LIN {X 0,Y 230.328,Z 772.05,A -85,B 0,C 180,E1 -20406.395,E2 -20406.395} C_VEL
LIN {X 0,Y 229.138,Z 759.993,A -85,B 0,C 180,E1 -20407.932,E2 -20407.932} C_VEL
LIN {X 0,Y 227.349,Z 746.527,A -85,B 0,C 180,E1 -20409.296,E2 -20409.296} C_VEL
LIN {X 0,Y 224.848,Z 732.445,A -85,B 0,C 180,E1 -20410.367,E2 -20410.367} C_VEL
LIN {X 0,Y 224.753,Z 731.518,A -85,B 0,C 180,E1 -20410.477,E2 -20410.477} C_VEL
LIN {X 0,Y 225.974,Z 721.97,A -85,B 0,C 180,E1 -20414.606,E2 -20414.606} C_VEL
LIN {X 0,Y 227.437,Z 711.151,A -85,B 0,C 180,E1 -20419.316,E2 -20419.316} C_VEL
LIN {X 0,Y 227.799,Z 707.066,A -85,B 0,C 180,E1 -20421.127,E2 -20421.127} C_VEL
LIN {X 0,Y 227.341,Z 701.42,A -85,B 0,C 180,E1 -20423.79,E2 -20423.79} C_VEL
LIN {X 0,Y 225.605,Z 691.076,A -85,B 0,C 180,E1 -20428.938,E2 -20428.938} C_VEL
LIN {X 0,Y 224.604,Z 685.498,A -85,B 0,C 180,E1 -20431.794,E2 -20431.794} C_VEL
LIN {X 0,Y 221.937,Z 675.451,A -85,B 0,C 180,E1 -20437.278,E2 -20437.278} C_VEL
LIN {X 0,Y 221.276,Z 672.918,A -85,B 0,C 180,E1 -20438.793,E2 -20438.793} C_VEL
LIN {X 0,Y 221.288,Z 673.134,A -85,B 0,C 180,E1 -20439.08,E2 -20439.08} C_VEL
LIN {X 0,Y 225.275,Z 684.524,A -85,B 0,C 180,E1 -20440.789,E2 -20440.789} C_VEL
LIN {X 0,Y 228.656,Z 695.212,A -85,B 0,C 180,E1 -20442.651,E2 -20442.651} C_VEL
LIN {X 0,Y 231.416,Z 705.742,A -85,B 0,C 180,E1 -20444.736,E2 -20444.736} C_VEL
LIN {X 0,Y 231.578,Z 706.808,A -85,B 0,C 180,E1 -20444.95,E2 -20444.95} C_VEL
LIN {X 0,Y 229.57,Z 717.919,A -85,B 0,C 180,E1 -20447.138,E2 -20447.138} C_VEL
LIN {X 0,Y 227.893,Z 726.962,A -85,B 0,C 180,E1 -20449.361,E2 -20449.361} C_VEL
LIN {X 0,Y 226.116,Z 735.343,A -85,B 0,C 180,E1 -20451.9,E2 -20451.9} C_VEL
LIN {X 0,Y 224.502,Z 742.894,A -85,B 0,C 180,E1 -20454.792,E2 -20454.792} C_VEL
LIN {X 0,Y 223.525,Z 747.733,A -85,B 0,C 180,E1 -20457.098,E2 -20457.098} C_VEL
LIN {X 0,Y 222.474,Z 753.098,A -85,B 0,C 180,E1 -20460.362,E2 -20460.362} C_VEL
LIN {X 0,Y 221.947,Z 755.831,A -85,B 0,C 180,E1 -20462.569,E2 -20462.569} C_VEL
LIN {X 0,Y 221.622,Z 757.987,A -85,B 0,C 180,E1 -20464.808,E2 -20464.808} C_VEL
LIN {X 0,Y 221.54,Z 759.729,A -85,B 0,C 180,E1 -20467.526,E2 -20467.526} C_VEL
LIN {X 0,Y 221.871,Z 760.631,A -85,B 0,C 180,E1 -20470.516,E2 -20470.516} C_VEL
LIN {X 0,Y 222.756,Z 760.329,A -85,B 0,C 180,E1 -20473.957,E2 -20473.957} C_VEL
LIN {X 0,Y 223.638,Z 759.356,A -85,B 0,C 180,E1 -20476.286,E2 -20476.286} C_VEL
LIN {X 0,Y 225.52,Z 756.419,A -85,B 0,C 180,E1 -20479.898,E2 -20479.898} C_VEL
LIN {X 0,Y 227.153,Z 753.336,A -85,B 0,C 180,E1 -20482.401,E2 -20482.401} C_VEL
LIN {X 0,Y 229.082,Z 749.336,A -85,B 0,C 180,E1 -20484.857,E2 -20484.857} C_VEL
LIN {X 0,Y 231.336,Z 744.272,A -85,B 0,C 180,E1 -20487.28,E2 -20487.28} C_VEL
LIN {X 0,Y 233.865,Z 738.05,A -85,B 0,C 180,E1 -20489.641,E2 -20489.641} C_VEL
LIN {X 0,Y 236.623,Z 730.403,A -85,B 0,C 180,E1 -20491.971,E2 -20491.971} C_VEL
LIN {X 0,Y 239.577,Z 721.408,A -85,B 0,C 180,E1 -20494.152,E2 -20494.152} C_VEL
LIN {X 0,Y 239.995,Z 719.96,A -85,B 0,C 180,E1 -20494.456,E2 -20494.456} C_VEL
LIN {X 0,Y 239.14,Z 713.976,A -85,B 0,C 180,E1 -20496.166,E2 -20496.166} C_VEL
LIN {X 0,Y 236.776,Z 705.016,A -85,B 0,C 180,E1 -20498.678,E2 -20498.678} C_VEL
LIN {X 0,Y 233.522,Z 696.191,A -85,B 0,C 180,E1 -20501.124,E2 -20501.124} C_VEL
LIN {X 0,Y 229.459,Z 687.704,A -85,B 0,C 180,E1 -20503.542,E2 -20503.542} C_VEL
LIN {X 0,Y 226.423,Z 682.123,A -85,B 0,C 180,E1 -20505.163,E2 -20505.163} C_VEL
LIN {X 0,Y 224.367,Z 678.912,A -85,B 0,C 180,E1 -20506.178,E2 -20506.178} C_VEL
LIN {X 0,Y 223.667,Z 677.621,A -85,B 0,C 180,E1 -20506.542,E2 -20506.542} C_VEL
LIN {X 0,Y 221.78,Z 675.276,A -85,B 0,C 180,E1 -20507.417,E2 -20507.417} C_VEL
LIN {X 0,Y 221.062,Z 672.945,A -85,B 0,C 180,E1 -20507.958,E2 -20507.958} C_VEL
LIN {X 0,Y 221.24,Z 672.924,A -85,B 0,C 180,E1 -20510.861,E2 -20510.861} C_VEL
LIN {X 0,Y 221.293,Z 672.907,A -85,B 0,C 180,E1 -20512.702,E2 -20512.702} C_VEL
LIN {X 0,Y 221.516,Z 672.886,A -85,B 0,C 180,E1 -20518.182,E2 -20518.182} C_VEL
LIN {X 0,Y 221.516,Z 672.88,A -85,B 0,C 180,E1 -20521.818,E2 -20521.818} C_VEL
LIN {X 0,Y 221.309,Z 672.918,A -85,B 0,C 180,E1 -20527.298,E2 -20527.298} C_VEL
LIN {X 0,Y 221.11,Z 672.944,A -85,B 0,C 180,E1 -20530.995,E2 -20530.995} C_VEL
LIN {X 0,Y 221.02,Z 672.944,A -85,B 0,C 180,E1 -20536.63,E2 -20536.63} C_VEL
LIN {X 0,Y 220.948,Z 673.087,A -85,B 0,C 180,E1 -20541.947,E2 -20541.947} C_VEL
LIN {X 0,Y 221.61,Z 676.139,A -85,B 0,C 180,E1 -20546.359,E2 -20546.359} C_VEL
LIN {X 0,Y 222.496,Z 680.424,A -85,B 0,C 180,E1 -20551.476,E2 -20551.476} C_VEL
LIN {X 0,Y 223.333,Z 683.935,A -85,B 0,C 180,E1 -20555.095,E2 -20555.095} C_VEL
LIN {X 0,Y 224.157,Z 688.047,A -85,B 0,C 180,E1 -20558.834,E2 -20558.834} C_VEL
LIN {X 0,Y 224.93,Z 692.081,A -85,B 0,C 180,E1 -20562.168,E2 -20562.168} C_VEL
LIN {X 0,Y 224.511,Z 693.459,A -85,B 0,C 180,E1 -20563.107,E2 -20563.107} C_VEL
LIN {X 0,Y 222.094,Z 696.117,A -85,B 0,C 180,E1 -20564.563,E2 -20564.563} C_VEL
LIN {X 0,Y 219.629,Z 698.835,A -85,B 0,C 180,E1 -20566.046,E2 -20566.046} C_VEL
LIN {X 0,Y 219.18,Z 700.319,A -85,B 0,C 180,E1 -20567.012,E2 -20567.012} C_VEL
LIN {X 0,Y 219.597,Z 703.203,A -85,B 0,C 180,E1 -20569.033,E2 -20569.033} C_VEL
LIN {X 0,Y 220.976,Z 707.443,A -85,B 0,C 180,E1 -20569.757,E2 -20569.757} C_VEL
LIN {X 0,Y 221.732,Z 709.798,A -85,B 0,C 180,E1 -20570.174,E2 -20570.174} C_VEL
LIN {X 0,Y 224.611,Z 722.385,A -85,B 0,C 180,E1 -20572.15,E2 -20572.15} C_VEL
LIN {X 0,Y 226.492,Z 736.93,A -85,B 0,C 180,E1 -20574.426,E2 -20574.426} C_VEL
LIN {X 0,Y 226.964,Z 748.451,A -85,B 0,C 180,E1 -20576.31,E2 -20576.31} C_VEL
LIN {X 0,Y 226.482,Z 760.232,A -85,B 0,C 180,E1 -20578.422,E2 -20578.422} C_VEL
LIN {X 0,Y 225.182,Z 771.012,A -85,B 0,C 180,E1 -20580.589,E2 -20580.589} C_VEL
LIN {X 0,Y 223.216,Z 780.783,A -85,B 0,C 180,E1 -20582.835,E2 -20582.835} C_VEL
LIN {X 0,Y 221.932,Z 786.81,A -85,B 0,C 180,E1 -20584.438,E2 -20584.438} C_VEL
LIN {X 0,Y 221.121,Z 796.098,A -85,B 0,C 180,E1 -20585.844,E2 -20585.844} C_VEL
LIN {X 0,Y 218.923,Z 807.176,A -85,B 0,C 180,E1 -20587.838,E2 -20587.838} C_VEL
LIN {X 0,Y 217.03,Z 816.687,A -85,B 0,C 180,E1 -20590.013,E2 -20590.013} C_VEL
LIN {X 0,Y 215.729,Z 823.747,A -85,B 0,C 180,E1 -20591.971,E2 -20591.971} C_VEL
LIN {X 0,Y 214.068,Z 831.966,A -85,B 0,C 180,E1 -20594.772,E2 -20594.772} C_VEL
LIN {X 0,Y 212.846,Z 838.572,A -85,B 0,C 180,E1 -20597.606,E2 -20597.606} C_VEL
LIN {X 0,Y 212.118,Z 843.817,A -85,B 0,C 180,E1 -20600.463,E2 -20600.463} C_VEL
LIN {X 0,Y 211.718,Z 847.843,A -85,B 0,C 180,E1 -20603.327,E2 -20603.327} C_VEL
LIN {X 0,Y 211.566,Z 850.772,A -85,B 0,C 180,E1 -20606.19,E2 -20606.19} C_VEL
LIN {X 0,Y 211.618,Z 852.149,A -85,B 0,C 180,E1 -20608.096,E2 -20608.096} C_VEL
LIN {X 0,Y 211.718,Z 853.102,A -85,B 0,C 180,E1 -20609.999,E2 -20609.999} C_VEL
LIN {X 0,Y 211.582,Z 853.643,A -85,B 0,C 180,E1 -20611.902,E2 -20611.902} C_VEL
LIN {X 0,Y 211.507,Z 853.693,A -85,B 0,C 180,E1 -20614.548,E2 -20614.548} C_VEL
LIN {X 0,Y 211.769,Z 852.796,A -85,B 0,C 180,E1 -20617.627,E2 -20617.627} C_VEL
LIN {X 0,Y 212.753,Z 850.263,A -85,B 0,C 180,E1 -20621.431,E2 -20621.431} C_VEL
LIN {X 0,Y 213.945,Z 847.262,A -85,B 0,C 180,E1 -20624.262,E2 -20624.262} C_VEL
LIN {X 0,Y 215.748,Z 843.249,A -85,B 0,C 180,E1 -20627.047,E2 -20627.047} C_VEL
LIN {X 0,Y 218.124,Z 838.128,A -85,B 0,C 180,E1 -20629.773,E2 -20629.773} C_VEL
LIN {X 0,Y 221.012,Z 831.011,A -85,B 0,C 180,E1 -20632.753,E2 -20632.753} C_VEL
LIN {X 0,Y 224.587,Z 822.54,A -85,B 0,C 180,E1 -20635.484,E2 -20635.484} C_VEL
LIN {X 0,Y 227.743,Z 814.382,A -85,B 0,C 180,E1 -20637.572,E2 -20637.572} C_VEL
LIN {X 0,Y 231.693,Z 803.348,A -85,B 0,C 180,E1 -20639.781,E2 -20639.781} C_VEL
LIN {X 0,Y 234.219,Z 792.567,A -85,B 0,C 180,E1 -20641.674,E2 -20641.674} C_VEL
LIN {X 0,Y 236.122,Z 782.049,A -85,B 0,C 180,E1 -20643.197,E2 -20643.197} C_VEL
LIN {X 0,Y 236.663,Z 772.17,A -85,B 0,C 180,E1 -20644.583,E2 -20644.583} C_VEL
LIN {X 0,Y 235.936,Z 759.615,A -85,B 0,C 180,E1 -20646.321,E2 -20646.321} C_VEL
LIN {X 0,Y 233.902,Z 747.598,A -85,B 0,C 180,E1 -20648.007,E2 -20648.007} C_VEL
LIN {X 0,Y 231.196,Z 736.83,A -85,B 0,C 180,E1 -20649.669,E2 -20649.669} C_VEL
LIN {X 0,Y 232.487,Z 726.541,A -85,B 0,C 180,E1 -20652.996,E2 -20652.996} C_VEL
LIN {X 0,Y 231.85,Z 720.918,A -85,B 0,C 180,E1 -20655.797,E2 -20655.797} C_VEL
LIN {X 0,Y 231.289,Z 715.047,A -85,B 0,C 180,E1 -20659.432,E2 -20659.432} C_VEL
LIN {X 0,Y 231.206,Z 712.321,A -85,B 0,C 180,E1 -20661.455,E2 -20661.455} C_VEL
LIN {X 0,Y 230.48,Z 709.689,A -85,B 0,C 180,E1 -20664.594,E2 -20664.594} C_VEL
LIN {X 0,Y 229.895,Z 708.666,A -85,B 0,C 180,E1 -20666.614,E2 -20666.614} C_VEL
LIN {X 0,Y 229.073,Z 707.669,A -85,B 0,C 180,E1 -20670.601,E2 -20670.601} C_VEL
LIN {X 0,Y 228.738,Z 707.718,A -85,B 0,C 180,E1 -20674.522,E2 -20674.522} C_VEL
LIN {X 0,Y 228.636,Z 708.866,A -85,B 0,C 180,E1 -20678.354,E2 -20678.354} C_VEL
LIN {X 0,Y 228.851,Z 710.877,A -85,B 0,C 180,E1 -20682.173,E2 -20682.173} C_VEL
LIN {X 0,Y 229.226,Z 713.608,A -85,B 0,C 180,E1 -20685.801,E2 -20685.801} C_VEL
LIN {X 0,Y 229.717,Z 717.073,A -85,B 0,C 180,E1 -20689.422,E2 -20689.422} C_VEL
LIN {X 0,Y 229.877,Z 720.218,A -85,B 0,C 180,E1 -20692.092,E2 -20692.092} C_VEL
LIN {X 0,Y 230.134,Z 724.883,A -85,B 0,C 180,E1 -20695.621,E2 -20695.621} C_VEL
LIN {X 0,Y 229.631,Z 729.151,A -85,B 0,C 180,E1 -20698.246,E2 -20698.246} C_VEL
LIN {X 0,Y 228.414,Z 733.521,A -85,B 0,C 180,E1 -20700.496,E2 -20700.496} C_VEL
LIN {X 0,Y 232.203,Z 745.97,A -85,B 0,C 180,E1 -20702.837,E2 -20702.837} C_VEL
LIN {X 0,Y 234.434,Z 755.353,A -85,B 0,C 180,E1 -20704.552,E2 -20704.552} C_VEL
LIN {X 0,Y 235.853,Z 765.803,A -85,B 0,C 180,E1 -20706.416,E2 -20706.416} C_VEL
LIN {X 0,Y 236.335,Z 776.14,A -85,B 0,C 180,E1 -20708.28,E2 -20708.28} C_VEL
LIN {X 0,Y 235.852,Z 784.869,A -85,B 0,C 180,E1 -20709.909,E2 -20709.909} C_VEL
LIN {X 0,Y 232.364,Z 795.916,A -85,B 0,C 180,E1 -20711.78,E2 -20711.78} C_VEL
LIN {X 0,Y 228.84,Z 805.569,A -85,B 0,C 180,E1 -20713.84,E2 -20713.84} C_VEL
LIN {X 0,Y 225.195,Z 814.647,A -85,B 0,C 180,E1 -20716.312,E2 -20716.312} C_VEL
LIN {X 0,Y 221.901,Z 822.242,A -85,B 0,C 180,E1 -20718.942,E2 -20718.942} C_VEL
LIN {X 0,Y 218.696,Z 829.135,A -85,B 0,C 180,E1 -20722.069,E2 -20722.069} C_VEL
LIN {X 0,Y 216.25,Z 834.03,A -85,B 0,C 180,E1 -20724.992,E2 -20724.992} C_VEL
LIN {X 0,Y 214.504,Z 837.523,A -85,B 0,C 180,E1 -20727.797,E2 -20727.797} C_VEL
LIN {X 0,Y 213.038,Z 840.245,A -85,B 0,C 180,E1 -20730.941,E2 -20730.941} C_VEL
LIN {X 0,Y 211.884,Z 841.91,A -85,B 0,C 180,E1 -20734.324,E2 -20734.324} C_VEL
LIN {X 0,Y 211.326,Z 842.306,A -85,B 0,C 180,E1 -20737.048,E2 -20737.048} C_VEL
LIN {X 0,Y 211.039,Z 841.827,A -85,B 0,C 180,E1 -20740.011,E2 -20740.011} C_VEL
LIN {X 0,Y 210.988,Z 840.439,A -85,B 0,C 180,E1 -20742.879,E2 -20742.879} C_VEL
LIN {X 0,Y 211.269,Z 838.167,A -85,B 0,C 180,E1 -20745.689,E2 -20745.689} C_VEL
LIN {X 0,Y 211.796,Z 835.033,A -85,B 0,C 180,E1 -20748.422,E2 -20748.422} C_VEL
LIN {X 0,Y 212.665,Z 829.806,A -85,B 0,C 180,E1 -20751.79,E2 -20751.79} C_VEL
LIN {X 0,Y 213.775,Z 824.373,A -85,B 0,C 180,E1 -20754.467,E2 -20754.467} C_VEL
LIN {X 0,Y 215.097,Z 817.661,A -85,B 0,C 180,E1 -20757.121,E2 -20757.121} C_VEL
LIN {X 0,Y 216.865,Z 809.387,A -85,B 0,C 180,E1 -20759.748,E2 -20759.748} C_VEL
LIN {X 0,Y 218.899,Z 799.547,A -85,B 0,C 180,E1 -20762.256,E2 -20762.256} C_VEL
LIN {X 0,Y 220.888,Z 789.374,A -85,B 0,C 180,E1 -20764.314,E2 -20764.314} C_VEL
LIN {X 0,Y 222.863,Z 778.099,A -85,B 0,C 180,E1 -20766.137,E2 -20766.137} C_VEL
LIN {X 0,Y 223.511,Z 772.868,A -85,B 0,C 180,E1 -20766.86,E2 -20766.86} C_VEL
LIN {X 0,Y 222.448,Z 761.406,A -85,B 0,C 180,E1 -20768.392,E2 -20768.392} C_VEL
LIN {X 0,Y 220.648,Z 747.49,A -85,B 0,C 180,E1 -20769.877,E2 -20769.877} C_VEL
LIN {X 0,Y 218.265,Z 733.565,A -85,B 0,C 180,E1 -20771.002,E2 -20771.002} C_VEL
LIN {X 0,Y 218.02,Z 731.6,A -85,B 0,C 180,E1 -20771.196,E2 -20771.196} C_VEL
LIN {X 0,Y 219.476,Z 720.534,A -85,B 0,C 180,E1 -20776.105,E2 -20776.105} C_VEL
LIN {X 0,Y 220.881,Z 710.592,A -85,B 0,C 180,E1 -20780.525,E2 -20780.525} C_VEL
LIN {X 0,Y 220.857,Z 705.961,A -85,B 0,C 180,E1 -20782.688,E2 -20782.688} C_VEL
LIN {X 0,Y 220.062,Z 700.469,A -85,B 0,C 180,E1 -20785.422,E2 -20785.422} C_VEL
LIN {X 0,Y 218.658,Z 691.492,A -85,B 0,C 180,E1 -20790.001,E2 -20790.001} C_VEL
LIN {X 0,Y 217.524,Z 686.335,A -85,B 0,C 180,E1 -20792.779,E2 -20792.779} C_VEL
LIN {X 0,Y 214.875,Z 676.124,A -85,B 0,C 180,E1 -20798.583,E2 -20798.583} C_VEL
LIN {X 0,Y 218.663,Z 686.527,A -85,B 0,C 180,E1 -20800.255,E2 -20800.255} C_VEL
LIN {X 0,Y 221.863,Z 696.753,A -85,B 0,C 180,E1 -20802.115,E2 -20802.115} C_VEL
LIN {X 0,Y 224.351,Z 706.152,A -85,B 0,C 180,E1 -20804.051,E2 -20804.051} C_VEL
LIN {X 0,Y 224.806,Z 708.137,A -85,B 0,C 180,E1 -20804.484,E2 -20804.484} C_VEL
LIN {X 0,Y 222.769,Z 719.101,A -85,B 0,C 180,E1 -20806.716,E2 -20806.716} C_VEL
LIN {X 0,Y 220.991,Z 728.204,A -85,B 0,C 180,E1 -20809.025,E2 -20809.025} C_VEL
LIN {X 0,Y 219.184,Z 736.385,A -85,B 0,C 180,E1 -20811.586,E2 -20811.586} C_VEL
LIN {X 0,Y 217.664,Z 743.353,A -85,B 0,C 180,E1 -20814.311,E2 -20814.311} C_VEL
LIN {X 0,Y 216.482,Z 748.935,A -85,B 0,C 180,E1 -20817.034,E2 -20817.034} C_VEL
LIN {X 0,Y 215.415,Z 754.236,A -85,B 0,C 180,E1 -20820.378,E2 -20820.378} C_VEL
LIN {X 0,Y 214.711,Z 758.087,A -85,B 0,C 180,E1 -20823.811,E2 -20823.811} C_VEL
LIN {X 0,Y 214.511,Z 759.903,A -85,B 0,C 180,E1 -20826.139,E2 -20826.139} C_VEL
LIN {X 0,Y 214.584,Z 761.084,A -85,B 0,C 180,E1 -20828.484,E2 -20828.484} C_VEL
LIN {X 0,Y 214.997,Z 761.714,A -85,B 0,C 180,E1 -20831.25,E2 -20831.25} C_VEL
LIN {X 0,Y 215.815,Z 761.434,A -85,B 0,C 180,E1 -20834.24,E2 -20834.24} C_VEL
LIN {X 0,Y 217.442,Z 759.622,A -85,B 0,C 180,E1 -20838.022,E2 -20838.022} C_VEL
LIN {X 0,Y 218.803,Z 757.543,A -85,B 0,C 180,E1 -20840.434,E2 -20840.434} C_VEL
LIN {X 0,Y 220.429,Z 754.7,A -85,B 0,C 180,E1 -20842.853,E2 -20842.853} C_VEL
LIN {X 0,Y 222.881,Z 749.89,A -85,B 0,C 180,E1 -20845.865,E2 -20845.865} C_VEL
LIN {X 0,Y 225.865,Z 743.511,A -85,B 0,C 180,E1 -20848.859,E2 -20848.859} C_VEL
LIN {X 0,Y 228.929,Z 736.062,A -85,B 0,C 180,E1 -20851.523,E2 -20851.523} C_VEL
LIN {X 0,Y 232.04,Z 727.593,A -85,B 0,C 180,E1 -20853.904,E2 -20853.904} C_VEL
LIN {X 0,Y 233.771,Z 722.459,A -85,B 0,C 180,E1 -20855.109,E2 -20855.109} C_VEL
LIN {X 0,Y 233.299,Z 717.909,A -85,B 0,C 180,E1 -20856.475,E2 -20856.475} C_VEL
LIN {X 0,Y 231.421,Z 709.596,A -85,B 0,C 180,E1 -20858.978,E2 -20858.978} C_VEL
LIN {X 0,Y 228.417,Z 700.69,A -85,B 0,C 180,E1 -20861.617,E2 -20861.617} C_VEL
LIN {X 0,Y 224.796,Z 692.52,A -85,B 0,C 180,E1 -20864.124,E2 -20864.124} C_VEL
LIN {X 0,Y 219.847,Z 683.358,A -85,B 0,C 180,E1 -20867.069,E2 -20867.069} C_VEL
LIN {X 0,Y 218.223,Z 681.207,A -85,B 0,C 180,E1 -20867.917,E2 -20867.917} C_VEL
LIN {X 0,Y 216.942,Z 678.699,A -85,B 0,C 180,E1 -20868.674,E2 -20868.674} C_VEL
LIN {X 0,Y 214.922,Z 676.297,A -85,B 0,C 180,E1 -20869.71,E2 -20869.71} C_VEL
LIN {X 0,Y 214.158,Z 673.81,A -85,B 0,C 180,E1 -20870.35,E2 -20870.35} C_VEL
LIN {X 0,Y 214.231,Z 673.786,A -85,B 0,C 180,E1 -20872.46,E2 -20872.46} C_VEL
LIN {X 0,Y 214.449,Z 673.765,A -85,B 0,C 180,E1 -20878.122,E2 -20878.122} C_VEL
LIN {X 0,Y 214.553,Z 673.748,A -85,B 0,C 180,E1 -20880,E2 -20880} C_VEL
LIN {X 0,Y 214.449,Z 673.761,A -85,B 0,C 180,E1 -20881.878,E2 -20881.878} C_VEL
LIN {X 0,Y 214.244,Z 673.795,A -85,B 0,C 180,E1 -20887.54,E2 -20887.54} C_VEL
LIN {X 0,Y 214.027,Z 673.824,A -85,B 0,C 180,E1 -20891.363,E2 -20891.363} C_VEL
LIN {X 0,Y 213.937,Z 673.834,A -85,B 0,C 180,E1 -20895.237,E2 -20895.237} C_VEL
LIN {X 0,Y 213.872,Z 673.926,A -85,B 0,C 180,E1 -20899.185,E2 -20899.185} C_VEL
LIN {X 0,Y 214.409,Z 676.374,A -85,B 0,C 180,E1 -20903.392,E2 -20903.392} C_VEL
LIN {X 0,Y 215.165,Z 679.831,A -85,B 0,C 180,E1 -20908.125,E2 -20908.125} C_VEL
LIN {X 0,Y 215.874,Z 683.285,A -85,B 0,C 180,E1 -20912.171,E2 -20912.171} C_VEL
LIN {X 0,Y 216.946,Z 687.826,A -85,B 0,C 180,E1 -20916.82,E2 -20916.82} C_VEL
LIN {X 0,Y 217.905,Z 692.785,A -85,B 0,C 180,E1 -20921.185,E2 -20921.185} C_VEL
LIN {X 0,Y 218.754,Z 697.625,A -85,B 0,C 180,E1 -20925.024,E2 -20925.024} C_VEL
LIN {X 0,Y 219.18,Z 700.319,A -85,B 0,C 180,E1 -20927.012,E2 -20927.012} C_VEL
LIN {X 0,Y 219.338,Z 702.214,A -85,B 0,C 180,E1 -20927.883,E2 -20927.883} C_VEL
LIN {X 0,Y 219.415,Z 705.738,A -85,B 0,C 180,E1 -20928.755,E2 -20928.755} C_VEL
LIN {X 0,Y 219.347,Z 711.784,A -85,B 0,C 180,E1 -20929.648,E2 -20929.648} C_VEL
LIN {X 0,Y 219.455,Z 725.409,A -85,B 0,C 180,E1 -20931.178,E2 -20931.178} C_VEL
LIN {X 0,Y 219.615,Z 727.215,A -85,B 0,C 180,E1 -20931.459,E2 -20931.459} C_VEL
LIN {X 0,Y 220.866,Z 740.35,A -85,B 0,C 180,E1 -20933.697,E2 -20933.697} C_VEL
LIN {X 0,Y 220.932,Z 752.132,A -85,B 0,C 180,E1 -20935.801,E2 -20935.801} C_VEL
LIN {X 0,Y 219.902,Z 764.307,A -85,B 0,C 180,E1 -20938.174,E2 -20938.174} C_VEL
LIN {X 0,Y 218.38,Z 774.032,A -85,B 0,C 180,E1 -20940.335,E2 -20940.335} C_VEL
LIN {X 0,Y 215.94,Z 784.039,A -85,B 0,C 180,E1 -20942.893,E2 -20942.893} C_VEL
LIN {X 0,Y 215.038,Z 788.104,A -85,B 0,C 180,E1 -20944.078,E2 -20944.078} C_VEL
LIN {X 0,Y 214.357,Z 795.724,A -85,B 0,C 180,E1 -20945.289,E2 -20945.289} C_VEL
LIN {X 0,Y 212.09,Z 806.828,A -85,B 0,C 180,E1 -20947.342,E2 -20947.342} C_VEL
LIN {X 0,Y 210.089,Z 816.49,A -85,B 0,C 180,E1 -20949.614,E2 -20949.614} C_VEL
LIN {X 0,Y 208.587,Z 824.185,A -85,B 0,C 180,E1 -20951.84,E2 -20951.84} C_VEL
LIN {X 0,Y 206.913,Z 832.296,A -85,B 0,C 180,E1 -20954.737,E2 -20954.737} C_VEL
LIN {X 0,Y 205.867,Z 837.8,A -85,B 0,C 180,E1 -20957.178,E2 -20957.178} C_VEL
LIN {X 0,Y 205.096,Z 843.16,A -85,B 0,C 180,E1 -20960.134,E2 -20960.134} C_VEL
LIN {X 0,Y 204.656,Z 847.295,A -85,B 0,C 180,E1 -20963.096,E2 -20963.096} C_VEL
LIN {X 0,Y 204.475,Z 850.321,A -85,B 0,C 180,E1 -20966.057,E2 -20966.057} C_VEL
LIN {X 0,Y 204.533,Z 851.788,A -85,B 0,C 180,E1 -20968.03,E2 -20968.03} C_VEL
LIN {X 0,Y 204.628,Z 852.783,A -85,B 0,C 180,E1 -20969.999,E2 -20969.999} C_VEL
LIN {X 0,Y 204.496,Z 853.368,A -85,B 0,C 180,E1 -20971.968,E2 -20971.968} C_VEL
LIN {X 0,Y 204.412,Z 853.549,A -85,B 0,C 180,E1 -20974.386,E2 -20974.386} C_VEL
LIN {X 0,Y 204.708,Z 852.715,A -85,B 0,C 180,E1 -20977.892,E2 -20977.892} C_VEL
LIN {X 0,Y 205.787,Z 850.299,A -85,B 0,C 180,E1 -20981.823,E2 -20981.823} C_VEL
LIN {X 0,Y 207.034,Z 847.395,A -85,B 0,C 180,E1 -20984.748,E2 -20984.748} C_VEL
LIN {X 0,Y 208.97,Z 843.517,A -85,B 0,C 180,E1 -20987.618,E2 -20987.618} C_VEL
LIN {X 0,Y 211.472,Z 838.551,A -85,B 0,C 180,E1 -20990.422,E2 -20990.422} C_VEL
LIN {X 0,Y 214.406,Z 831.876,A -85,B 0,C 180,E1 -20993.391,E2 -20993.391} C_VEL
LIN {X 0,Y 218.253,Z 823.334,A -85,B 0,C 180,E1 -20996.279,E2 -20996.279} C_VEL
LIN {X 0,Y 221.538,Z 815.442,A -85,B 0,C 180,E1 -20998.414,E2 -20998.414} C_VEL
LIN {X 0,Y 225.319,Z 805.914,A -85,B 0,C 180,E1 -21000.453,E2 -21000.453} C_VEL
LIN {X 0,Y 228.395,Z 794.369,A -85,B 0,C 180,E1 -21002.58,E2 -21002.58} C_VEL
LIN {X 0,Y 230.639,Z 783.38,A -85,B 0,C 180,E1 -21004.254,E2 -21004.254} C_VEL
LIN {X 0,Y 231.404,Z 772.262,A -85,B 0,C 180,E1 -21005.923,E2 -21005.923} C_VEL
LIN {X 0,Y 230.829,Z 760.451,A -85,B 0,C 180,E1 -21007.663,E2 -21007.663} C_VEL
LIN {X 0,Y 228.95,Z 748.392,A -85,B 0,C 180,E1 -21009.489,E2 -21009.489} C_VEL
LIN {X 0,Y 226.033,Z 736.698,A -85,B 0,C 180,E1 -21011.466,E2 -21011.466} C_VEL
LIN {X 0,Y 227.046,Z 729.932,A -85,B 0,C 180,E1 -21013.796,E2 -21013.796} C_VEL
LIN {X 0,Y 226.387,Z 724.06,A -85,B 0,C 180,E1 -21016.923,E2 -21016.923} C_VEL
LIN {X 0,Y 226.016,Z 717.926,A -85,B 0,C 180,E1 -21021.019,E2 -21021.019} C_VEL
LIN {X 0,Y 226.015,Z 717.257,A -85,B 0,C 180,E1 -21021.544,E2 -21021.544} C_VEL
LIN {X 0,Y 225.388,Z 714.94,A -85,B 0,C 180,E1 -21024.165,E2 -21024.165} C_VEL
LIN {X 0,Y 225.023,Z 713.904,A -85,B 0,C 180,E1 -21025.793,E2 -21025.793} C_VEL
LIN {X 0,Y 223.942,Z 712.613,A -85,B 0,C 180,E1 -21029.859,E2 -21029.859} C_VEL
LIN {X 0,Y 223.466,Z 712.381,A -85,B 0,C 180,E1 -21033.877,E2 -21033.877} C_VEL
LIN {X 0,Y 223.225,Z 713.295,A -85,B 0,C 180,E1 -21037.802,E2 -21037.802} C_VEL
LIN {X 0,Y 223.297,Z 715.08,A -85,B 0,C 180,E1 -21041.655,E2 -21041.655} C_VEL
LIN {X 0,Y 223.544,Z 717.66,A -85,B 0,C 180,E1 -21045.433,E2 -21045.433} C_VEL
LIN {X 0,Y 223.904,Z 720.987,A -85,B 0,C 180,E1 -21049.144,E2 -21049.144} C_VEL
LIN {X 0,Y 224.068,Z 722.939,A -85,B 0,C 180,E1 -21050.977,E2 -21050.977} C_VEL
LIN {X 0,Y 224.149,Z 727.452,A -85,B 0,C 180,E1 -21054.602,E2 -21054.602} C_VEL
LIN {X 0,Y 223.97,Z 730.029,A -85,B 0,C 180,E1 -21056.402,E2 -21056.402} C_VEL
LIN {X 0,Y 223.205,Z 733.778,A -85,B 0,C 180,E1 -21058.553,E2 -21058.553} C_VEL
LIN {X 0,Y 226.851,Z 745.79,A -85,B 0,C 180,E1 -21061.054,E2 -21061.054} C_VEL
LIN {X 0,Y 229.284,Z 757.104,A -85,B 0,C 180,E1 -21063.277,E2 -21063.277} C_VEL
LIN {X 0,Y 230.648,Z 768.646,A -85,B 0,C 180,E1 -21065.464,E2 -21065.464} C_VEL
LIN {X 0,Y 230.739,Z 779.601,A -85,B 0,C 180,E1 -21067.578,E2 -21067.578} C_VEL
LIN {X 0,Y 230.139,Z 786.571,A -85,B 0,C 180,E1 -21068.957,E2 -21068.957} C_VEL
LIN {X 0,Y 226.732,Z 796.671,A -85,B 0,C 180,E1 -21070.718,E2 -21070.718} C_VEL
LIN {X 0,Y 222.733,Z 806.896,A -85,B 0,C 180,E1 -21072.992,E2 -21072.992} C_VEL
LIN {X 0,Y 218.849,Z 815.871,A -85,B 0,C 180,E1 -21075.553,E2 -21075.553} C_VEL
LIN {X 0,Y 215.993,Z 822.015,A -85,B 0,C 180,E1 -21077.76,E2 -21077.76} C_VEL
LIN {X 0,Y 212.632,Z 828.773,A -85,B 0,C 180,E1 -21080.812,E2 -21080.812} C_VEL
LIN {X 0,Y 210.114,Z 833.575,A -85,B 0,C 180,E1 -21083.664,E2 -21083.664} C_VEL
LIN {X 0,Y 207.792,Z 837.763,A -85,B 0,C 180,E1 -21087.058,E2 -21087.058} C_VEL
LIN {X 0,Y 206.006,Z 840.781,A -85,B 0,C 180,E1 -21090.779,E2 -21090.779} C_VEL
LIN {X 0,Y 204.723,Z 842.286,A -85,B 0,C 180,E1 -21094.525,E2 -21094.525} C_VEL
LIN {X 0,Y 204.059,Z 842.379,A -85,B 0,C 180,E1 -21098.311,E2 -21098.311} C_VEL
LIN {X 0,Y 203.877,Z 841.561,A -85,B 0,C 180,E1 -21100.917,E2 -21100.917} C_VEL
LIN {X 0,Y 204.044,Z 838.969,A -85,B 0,C 180,E1 -21104.916,E2 -21104.916} C_VEL
LIN {X 0,Y 204.532,Z 836.126,A -85,B 0,C 180,E1 -21107.698,E2 -21107.698} C_VEL
LIN {X 0,Y 205.224,Z 832.037,A -85,B 0,C 180,E1 -21110.664,E2 -21110.664} C_VEL
LIN {X 0,Y 206.461,Z 825.843,A -85,B 0,C 180,E1 -21114.045,E2 -21114.045} C_VEL
LIN {X 0,Y 207.672,Z 819.835,A -85,B 0,C 180,E1 -21116.639,E2 -21116.639} C_VEL
LIN {X 0,Y 209.493,Z 811.583,A -85,B 0,C 180,E1 -21119.51,E2 -21119.51} C_VEL
LIN {X 0,Y 211.37,Z 802.631,A -85,B 0,C 180,E1 -21121.99,E2 -21121.99} C_VEL
LIN {X 0,Y 213.582,Z 791.966,A -85,B 0,C 180,E1 -21124.355,E2 -21124.355} C_VEL
LIN {X 0,Y 215.741,Z 780.381,A -85,B 0,C 180,E1 -21126.371,E2 -21126.371} C_VEL
LIN {X 0,Y 216.67,Z 773.685,A -85,B 0,C 180,E1 -21127.346,E2 -21127.346} C_VEL
LIN {X 0,Y 215.647,Z 761.904,A -85,B 0,C 180,E1 -21128.994,E2 -21128.994} C_VEL
LIN {X 0,Y 213.961,Z 748.23,A -85,B 0,C 180,E1 -21130.514,E2 -21130.514} C_VEL
LIN {X 0,Y 211.795,Z 735.31,A -85,B 0,C 180,E1 -21131.626,E2 -21131.626} C_VEL
LIN {X 0,Y 211.22,Z 731.878,A -85,B 0,C 180,E1 -21131.888,E2 -21131.888} C_VEL
LIN {X 0,Y 212.839,Z 720.291,A -85,B 0,C 180,E1 -21137.122,E2 -21137.122} C_VEL
LIN {X 0,Y 214.047,Z 712.187,A -85,B 0,C 180,E1 -21140.811,E2 -21140.811} C_VEL
LIN {X 0,Y 213.949,Z 706.812,A -85,B 0,C 180,E1 -21143.399,E2 -21143.399} C_VEL
LIN {X 0,Y 212.768,Z 699.499,A -85,B 0,C 180,E1 -21147.161,E2 -21147.161} C_VEL
LIN {X 0,Y 211.635,Z 691.997,A -85,B 0,C 180,E1 -21151.123,E2 -21151.123} C_VEL
LIN {X 0,Y 210.354,Z 687.194,A -85,B 0,C 180,E1 -21153.832,E2 -21153.832} C_VEL
LIN {X 0,Y 208.542,Z 679.781,A -85,B 0,C 180,E1 -21158.114,E2 -21158.114} C_VEL
LIN {X 0,Y 209.553,Z 681.188,A -85,B 0,C 180,E1 -21158.438,E2 -21158.438} C_VEL
LIN {X 0,Y 213.329,Z 692.548,A -85,B 0,C 180,E1 -21160.44,E2 -21160.44} C_VEL
LIN {X 0,Y 216.173,Z 702.165,A -85,B 0,C 180,E1 -21162.368,E2 -21162.368} C_VEL
LIN {X 0,Y 217.973,Z 709.528,A -85,B 0,C 180,E1 -21163.996,E2 -21163.996} C_VEL
LIN {X 0,Y 215.936,Z 720.436,A -85,B 0,C 180,E1 -21166.304,E2 -21166.304} C_VEL
LIN {X 0,Y 213.906,Z 730.192,A -85,B 0,C 180,E1 -21168.892,E2 -21168.892} C_VEL
LIN {X 0,Y 211.948,Z 738.884,A -85,B 0,C 180,E1 -21171.806,E2 -21171.806} C_VEL
LIN {X 0,Y 210.483,Z 745.286,A -85,B 0,C 180,E1 -21174.481,E2 -21174.481} C_VEL
LIN {X 0,Y 209.452,Z 750.059,A -85,B 0,C 180,E1 -21176.936,E2 -21176.936} C_VEL
LIN {X 0,Y 208.369,Z 755.342,A -85,B 0,C 180,E1 -21180.394,E2 -21180.394} C_VEL
LIN {X 0,Y 207.639,Z 759.18,A -85,B 0,C 180,E1 -21183.952,E2 -21183.952} C_VEL
LIN {X 0,Y 207.489,Z 761.646,A -85,B 0,C 180,E1 -21187.568,E2 -21187.568} C_VEL
LIN {X 0,Y 207.733,Z 762.533,A -85,B 0,C 180,E1 -21190.002,E2 -21190.002} C_VEL
LIN {X 0,Y 208.257,Z 762.801,A -85,B 0,C 180,E1 -21192.45,E2 -21192.45} C_VEL
LIN {X 0,Y 209.1,Z 762.371,A -85,B 0,C 180,E1 -21195.104,E2 -21195.104} C_VEL
LIN {X 0,Y 210.433,Z 760.995,A -85,B 0,C 180,E1 -21198.091,E2 -21198.091} C_VEL
LIN {X 0,Y 212.087,Z 758.705,A -85,B 0,C 180,E1 -21200.979,E2 -21200.979} C_VEL
LIN {X 0,Y 214.046,Z 755.495,A -85,B 0,C 180,E1 -21203.771,E2 -21203.771} C_VEL
LIN {X 0,Y 216.341,Z 751.307,A -85,B 0,C 180,E1 -21206.478,E2 -21206.478} C_VEL
LIN {X 0,Y 219.701,Z 744.577,A -85,B 0,C 180,E1 -21209.736,E2 -21209.736} C_VEL
LIN {X 0,Y 222.56,Z 738.078,A -85,B 0,C 180,E1 -21212.152,E2 -21212.152} C_VEL
LIN {X 0,Y 225.715,Z 729.965,A -85,B 0,C 180,E1 -21214.551,E2 -21214.551} C_VEL
LIN {X 0,Y 227.671,Z 724.327,A -85,B 0,C 180,E1 -21215.954,E2 -21215.954} C_VEL
LIN {X 0,Y 226.725,Z 717.557,A -85,B 0,C 180,E1 -21218.163,E2 -21218.163} C_VEL
LIN {X 0,Y 224.622,Z 709.239,A -85,B 0,C 180,E1 -21220.821,E2 -21220.821} C_VEL
LIN {X 0,Y 221.735,Z 701.21,A -85,B 0,C 180,E1 -21223.426,E2 -21223.426} C_VEL
LIN {X 0,Y 218.175,Z 693.335,A -85,B 0,C 180,E1 -21226.057,E2 -21226.057} C_VEL
LIN {X 0,Y 214.989,Z 687.719,A -85,B 0,C 180,E1 -21228.114,E2 -21228.114} C_VEL
LIN {X 0,Y 213.001,Z 684.245,A -85,B 0,C 180,E1 -21229.387,E2 -21229.387} C_VEL
LIN {X 0,Y 210.896,Z 680.909,A -85,B 0,C 180,E1 -21230.711,E2 -21230.711} C_VEL
LIN {X 0,Y 210.531,Z 679.891,A -85,B 0,C 180,E1 -21230.998,E2 -21230.998} C_VEL
LIN {X 0,Y 208.387,Z 677.825,A -85,B 0,C 180,E1 -21232.186,E2 -21232.186} C_VEL
LIN {X 0,Y 207.184,Z 674.983,A -85,B 0,C 180,E1 -21233.059,E2 -21233.059} C_VEL
LIN {X 0,Y 207.13,Z 674.672,A -85,B 0,C 180,E1 -21233.18,E2 -21233.18} C_VEL
LIN {X 0,Y 207.386,Z 674.644,A -85,B 0,C 180,E1 -21238.058,E2 -21238.058} C_VEL
LIN {X 0,Y 207.518,Z 674.624,A -85,B 0,C 180,E1 -21240,E2 -21240} C_VEL
LIN {X 0,Y 207.386,Z 674.641,A -85,B 0,C 180,E1 -21241.942,E2 -21241.942} C_VEL
LIN {X 0,Y 207.182,Z 674.672,A -85,B 0,C 180,E1 -21247.799,E2 -21247.799} C_VEL
LIN {X 0,Y 206.947,Z 674.701,A -85,B 0,C 180,E1 -21251.757,E2 -21251.757} C_VEL
LIN {X 0,Y 206.877,Z 674.723,A -85,B 0,C 180,E1 -21255.77,E2 -21255.77} C_VEL
LIN {X 0,Y 207.258,Z 676.664,A -85,B 0,C 180,E1 -21259.822,E2 -21259.822} C_VEL
LIN {X 0,Y 207.8,Z 679.171,A -85,B 0,C 180,E1 -21264.052,E2 -21264.052} C_VEL
LIN {X 0,Y 208.537,Z 682.649,A -85,B 0,C 180,E1 -21268.807,E2 -21268.807} C_VEL
LIN {X 0,Y 209.285,Z 686.133,A -85,B 0,C 180,E1 -21272.909,E2 -21272.909} C_VEL
LIN {X 0,Y 210.185,Z 690.097,A -85,B 0,C 180,E1 -21277.004,E2 -21277.004} C_VEL
LIN {X 0,Y 211.174,Z 695.355,A -85,B 0,C 180,E1 -21281.73,E2 -21281.73} C_VEL
LIN {X 0,Y 212.179,Z 701.2,A -85,B 0,C 180,E1 -21286.407,E2 -21286.407} C_VEL
LIN {X 0,Y 213.721,Z 705.332,A -85,B 0,C 180,E1 -21287.285,E2 -21287.285} C_VEL
LIN {X 0,Y 215.56,Z 708.407,A -85,B 0,C 180,E1 -21288.169,E2 -21288.169} C_VEL
LIN {X 0,Y 217.124,Z 713.716,A -85,B 0,C 180,E1 -21289.168,E2 -21289.168} C_VEL
LIN {X 0,Y 219.457,Z 725.753,A -85,B 0,C 180,E1 -21291.224,E2 -21291.224} C_VEL
LIN {X 0,Y 219.615,Z 727.215,A -85,B 0,C 180,E1 -21291.459,E2 -21291.459} C_VEL
LIN {X 0,Y 219.718,Z 732.499,A -85,B 0,C 180,E1 -21292.211,E2 -21292.211} C_VEL
LIN {X 0,Y 217.917,Z 741.67,A -85,B 0,C 180,E1 -21293.228,E2 -21293.228} C_VEL
LIN {X 0,Y 215.61,Z 750.315,A -85,B 0,C 180,E1 -21294.324,E2 -21294.324} C_VEL
LIN {X 0,Y 214.842,Z 755.144,A -85,B 0,C 180,E1 -21295.171,E2 -21295.171} C_VEL
LIN {X 0,Y 213.484,Z 766.878,A -85,B 0,C 180,E1 -21297.658,E2 -21297.658} C_VEL
LIN {X 0,Y 211.441,Z 776.966,A -85,B 0,C 180,E1 -21300.093,E2 -21300.093} C_VEL
LIN {X 0,Y 208.714,Z 786.992,A -85,B 0,C 180,E1 -21302.961,E2 -21302.961} C_VEL
LIN {X 0,Y 208.158,Z 789.326,A -85,B 0,C 180,E1 -21303.695,E2 -21303.695} C_VEL
LIN {X 0,Y 207.287,Z 796.705,A -85,B 0,C 180,E1 -21304.924,E2 -21304.924} C_VEL
LIN {X 0,Y 205.066,Z 807.581,A -85,B 0,C 180,E1 -21307.054,E2 -21307.054} C_VEL
LIN {X 0,Y 203.162,Z 816.283,A -85,B 0,C 180,E1 -21309.185,E2 -21309.185} C_VEL
LIN {X 0,Y 201.451,Z 824.614,A -85,B 0,C 180,E1 -21311.7,E2 -21311.7} C_VEL
LIN {X 0,Y 199.76,Z 832.606,A -85,B 0,C 180,E1 -21314.699,E2 -21314.699} C_VEL
LIN {X 0,Y 198.576,Z 838.996,A -85,B 0,C 180,E1 -21317.739,E2 -21317.739} C_VEL
LIN {X 0,Y 197.885,Z 844.03,A -85,B 0,C 180,E1 -21320.803,E2 -21320.803} C_VEL
LIN {X 0,Y 197.504,Z 847.883,A -85,B 0,C 180,E1 -21323.871,E2 -21323.871} C_VEL
LIN {X 0,Y 197.395,Z 849.84,A -85,B 0,C 180,E1 -21325.916,E2 -21325.916} C_VEL
LIN {X 0,Y 197.45,Z 851.374,A -85,B 0,C 180,E1 -21327.959,E2 -21327.959} C_VEL
LIN {X 0,Y 197.541,Z 852.454,A -85,B 0,C 180,E1 -21329.999,E2 -21329.999} C_VEL
LIN {X 0,Y 197.393,Z 853.088,A -85,B 0,C 180,E1 -21332.039,E2 -21332.039} C_VEL
LIN {X 0,Y 197.41,Z 853.193,A -85,B 0,C 180,E1 -21336.13,E2 -21336.13} C_VEL
LIN {X 0,Y 197.67,Z 852.634,A -85,B 0,C 180,E1 -21338.175,E2 -21338.175} C_VEL
LIN {X 0,Y 198.82,Z 850.335,A -85,B 0,C 180,E1 -21342.244,E2 -21342.244} C_VEL
LIN {X 0,Y 200.149,Z 847.557,A -85,B 0,C 180,E1 -21345.268,E2 -21345.268} C_VEL
LIN {X 0,Y 202.203,Z 843.799,A -85,B 0,C 180,E1 -21348.228,E2 -21348.228} C_VEL
LIN {X 0,Y 204.85,Z 838.96,A -85,B 0,C 180,E1 -21351.113,E2 -21351.113} C_VEL
LIN {X 0,Y 208.21,Z 831.998,A -85,B 0,C 180,E1 -21354.369,E2 -21354.369} C_VEL
LIN {X 0,Y 211.966,Z 824.232,A -85,B 0,C 180,E1 -21357.121,E2 -21357.121} C_VEL
LIN {X 0,Y 215.389,Z 816.547,A -85,B 0,C 180,E1 -21359.302,E2 -21359.302} C_VEL
LIN {X 0,Y 219.722,Z 806.257,A -85,B 0,C 180,E1 -21361.584,E2 -21361.584} C_VEL
LIN {X 0,Y 222.614,Z 796.275,A -85,B 0,C 180,E1 -21363.536,E2 -21363.536} C_VEL
LIN {X 0,Y 225.355,Z 784.337,A -85,B 0,C 180,E1 -21365.448,E2 -21365.448} C_VEL
LIN {X 0,Y 226.27,Z 773.177,A -85,B 0,C 180,E1 -21367.206,E2 -21367.206} C_VEL
LIN {X 0,Y 225.955,Z 762.108,A -85,B 0,C 180,E1 -21368.959,E2 -21368.959} C_VEL
LIN {X 0,Y 224.521,Z 751.284,A -85,B 0,C 180,E1 -21370.728,E2 -21370.728} C_VEL
LIN {X 0,Y 221.998,Z 740.191,A -85,B 0,C 180,E1 -21372.711,E2 -21372.711} C_VEL
LIN {X 0,Y 221.132,Z 736.444,A -85,B 0,C 180,E1 -21373.461,E2 -21373.461} C_VEL
LIN {X 0,Y 221.55,Z 734.228,A -85,B 0,C 180,E1 -21374.256,E2 -21374.256} C_VEL
LIN {X 0,Y 221.145,Z 729.092,A -85,B 0,C 180,E1 -21376.963,E2 -21376.963} C_VEL
LIN {X 0,Y 220.79,Z 723.752,A -85,B 0,C 180,E1 -21380.459,E2 -21380.459} C_VEL
LIN {X 0,Y 220.81,Z 722.185,A -85,B 0,C 180,E1 -21381.636,E2 -21381.636} C_VEL
LIN {X 0,Y 220.062,Z 719.356,A -85,B 0,C 180,E1 -21384.91,E2 -21384.91} C_VEL
LIN {X 0,Y 219.439,Z 718.294,A -85,B 0,C 180,E1 -21387.012,E2 -21387.012} C_VEL
LIN {X 0,Y 218.509,Z 717.243,A -85,B 0,C 180,E1 -21391.154,E2 -21391.154} C_VEL
LIN {X 0,Y 218.014,Z 717.304,A -85,B 0,C 180,E1 -21395.224,E2 -21395.224} C_VEL
LIN {X 0,Y 217.767,Z 718.499,A -85,B 0,C 180,E1 -21399.373,E2 -21399.373} C_VEL
LIN {X 0,Y 217.808,Z 720.456,A -85,B 0,C 180,E1 -21403.118,E2 -21403.118} C_VEL
LIN {X 0,Y 217.992,Z 723.295,A -85,B 0,C 180,E1 -21406.957,E2 -21406.957} C_VEL
LIN {X 0,Y 218.238,Z 726.87,A -85,B 0,C 180,E1 -21410.734,E2 -21410.734} C_VEL
LIN {X 0,Y 218.163,Z 731.324,A -85,B 0,C 180,E1 -21414.454,E2 -21414.454} C_VEL
LIN {X 0,Y 217.923,Z 734.087,A -85,B 0,C 180,E1 -21416.302,E2 -21416.302} C_VEL
LIN {X 0,Y 219.97,Z 739.758,A -85,B 0,C 180,E1 -21417.768,E2 -21417.768} C_VEL
LIN {X 0,Y 222.668,Z 750.035,A -85,B 0,C 180,E1 -21420.056,E2 -21420.056} C_VEL
LIN {X 0,Y 224.737,Z 762.094,A -85,B 0,C 180,E1 -21422.571,E2 -21422.571} C_VEL
LIN {X 0,Y 225.496,Z 773.64,A -85,B 0,C 180,E1 -21424.917,E2 -21424.917} C_VEL
LIN {X 0,Y 225.101,Z 783.578,A -85,B 0,C 180,E1 -21426.949,E2 -21426.949} C_VEL
LIN {X 0,Y 224.645,Z 787.845,A -85,B 0,C 180,E1 -21427.867,E2 -21427.867} C_VEL
LIN {X 0,Y 220.631,Z 798.758,A -85,B 0,C 180,E1 -21429.877,E2 -21429.877} C_VEL
LIN {X 0,Y 216.295,Z 809.114,A -85,B 0,C 180,E1 -21432.316,E2 -21432.316} C_VEL
LIN {X 0,Y 212.404,Z 817.427,A -85,B 0,C 180,E1 -21434.858,E2 -21434.858} C_VEL
LIN {X 0,Y 208.808,Z 824.527,A -85,B 0,C 180,E1 -21437.633,E2 -21437.633} C_VEL
LIN {X 0,Y 205.311,Z 830.934,A -85,B 0,C 180,E1 -21440.884,E2 -21440.884} C_VEL
LIN {X 0,Y 203.058,Z 834.8,A -85,B 0,C 180,E1 -21443.454,E2 -21443.454} C_VEL
LIN {X 0,Y 200.622,Z 838.811,A -85,B 0,C 180,E1 -21447.091,E2 -21447.091} C_VEL
LIN {X 0,Y 199.377,Z 840.687,A -85,B 0,C 180,E1 -21449.57,E2 -21449.57} C_VEL
LIN {X 0,Y 198.347,Z 841.962,A -85,B 0,C 180,E1 -21452.106,E2 -21452.106} C_VEL
LIN {X 0,Y 197.498,Z 842.683,A -85,B 0,C 180,E1 -21455.072,E2 -21455.072} C_VEL
LIN {X 0,Y 196.985,Z 842.512,A -85,B 0,C 180,E1 -21458.29,E2 -21458.29} C_VEL
LIN {X 0,Y 196.779,Z 841.411,A -85,B 0,C 180,E1 -21461.41,E2 -21461.41} C_VEL
LIN {X 0,Y 197.027,Z 838.483,A -85,B 0,C 180,E1 -21465.512,E2 -21465.512} C_VEL
LIN {X 0,Y 197.543,Z 835.442,A -85,B 0,C 180,E1 -21468.341,E2 -21468.341} C_VEL
LIN {X 0,Y 198.259,Z 831.345,A -85,B 0,C 180,E1 -21471.248,E2 -21471.248} C_VEL
LIN {X 0,Y 199.373,Z 826.095,A -85,B 0,C 180,E1 -21474.17,E2 -21474.17} C_VEL
LIN {X 0,Y 200.775,Z 819.381,A -85,B 0,C 180,E1 -21477.151,E2 -21477.151} C_VEL
LIN {X 0,Y 202.688,Z 811.017,A -85,B 0,C 180,E1 -21480.094,E2 -21480.094} C_VEL
LIN {X 0,Y 204.662,Z 801.942,A -85,B 0,C 180,E1 -21482.645,E2 -21482.645} C_VEL
LIN {X 0,Y 206.722,Z 792.299,A -85,B 0,C 180,E1 -21484.837,E2 -21484.837} C_VEL
LIN {X 0,Y 208.696,Z 782.192,A -85,B 0,C 180,E1 -21486.692,E2 -21486.692} C_VEL
LIN {X 0,Y 209.856,Z 774.469,A -85,B 0,C 180,E1 -21487.868,E2 -21487.868} C_VEL
LIN {X 0,Y 208.912,Z 762.75,A -85,B 0,C 180,E1 -21489.574,E2 -21489.574} C_VEL
LIN {X 0,Y 207.366,Z 749.717,A -85,B 0,C 180,E1 -21491.091,E2 -21491.091} C_VEL
LIN {X 0,Y 205.217,Z 736.367,A -85,B 0,C 180,E1 -21492.307,E2 -21492.307} C_VEL
LIN {X 0,Y 204.47,Z 732.069,A -85,B 0,C 180,E1 -21492.628,E2 -21492.628} C_VEL
LIN {X 0,Y 206.23,Z 720.039,A -85,B 0,C 180,E1 -21498.203,E2 -21498.203} C_VEL
LIN {X 0,Y 207.316,Z 712.489,A -85,B 0,C 180,E1 -21501.717,E2 -21501.717} C_VEL
LIN {X 0,Y 207.015,Z 707.641,A -85,B 0,C 180,E1 -21504.156,E2 -21504.156} C_VEL
LIN {X 0,Y 205.367,Z 696.683,A -85,B 0,C 180,E1 -21510.001,E2 -21510.001} C_VEL
LIN {X 0,Y 204.131,Z 690.986,A -85,B 0,C 180,E1 -21513.205,E2 -21513.205} C_VEL
LIN {X 0,Y 202.245,Z 683.435,A -85,B 0,C 180,E1 -21517.677,E2 -21517.677} C_VEL
LIN {X 0,Y 203.807,Z 685.396,A -85,B 0,C 180,E1 -21518.179,E2 -21518.179} C_VEL
LIN {X 0,Y 207.296,Z 696.33,A -85,B 0,C 180,E1 -21520.253,E2 -21520.253} C_VEL
LIN {X 0,Y 210.097,Z 706.512,A -85,B 0,C 180,E1 -21522.459,E2 -21522.459} C_VEL
LIN {X 0,Y 211.101,Z 710.832,A -85,B 0,C 180,E1 -21523.477,E2 -21523.477} C_VEL
LIN {X 0,Y 209.311,Z 720.52,A -85,B 0,C 180,E1 -21525.583,E2 -21525.583} C_VEL
LIN {X 0,Y 207.215,Z 730.49,A -85,B 0,C 180,E1 -21528.257,E2 -21528.257} C_VEL
LIN {X 0,Y 205.322,Z 738.601,A -85,B 0,C 180,E1 -21530.982,E2 -21530.982} C_VEL
LIN {X 0,Y 203.677,Z 745.61,A -85,B 0,C 180,E1 -21533.92,E2 -21533.92} C_VEL
LIN {X 0,Y 202.408,Z 751.171,A -85,B 0,C 180,E1 -21536.834,E2 -21536.834} C_VEL
LIN {X 0,Y 201.299,Z 756.447,A -85,B 0,C 180,E1 -21540.414,E2 -21540.414} C_VEL
LIN {X 0,Y 200.584,Z 760.27,A -85,B 0,C 180,E1 -21544.098,E2 -21544.098} C_VEL
LIN {X 0,Y 200.451,Z 762.077,A -85,B 0,C 180,E1 -21546.587,E2 -21546.587} C_VEL
LIN {X 0,Y 200.642,Z 763.405,A -85,B 0,C 180,E1 -21549.592,E2 -21549.592} C_VEL
LIN {X 0,Y 201.326,Z 763.866,A -85,B 0,C 180,E1 -21552.855,E2 -21552.855} C_VEL
LIN {X 0,Y 202.732,Z 763.063,A -85,B 0,C 180,E1 -21556.72,E2 -21556.72} C_VEL
LIN {X 0,Y 204.773,Z 760.758,A -85,B 0,C 180,E1 -21560.555,E2 -21560.555} C_VEL
LIN {X 0,Y 206.493,Z 758.292,A -85,B 0,C 180,E1 -21563.118,E2 -21563.118} C_VEL
LIN {X 0,Y 208.641,Z 754.799,A -85,B 0,C 180,E1 -21565.818,E2 -21565.818} C_VEL
LIN {X 0,Y 211.182,Z 750.327,A -85,B 0,C 180,E1 -21568.45,E2 -21568.45} C_VEL
LIN {X 0,Y 214.531,Z 743.66,A -85,B 0,C 180,E1 -21571.478,E2 -21571.478} C_VEL
LIN {X 0,Y 217.683,Z 736.666,A -85,B 0,C 180,E1 -21573.961,E2 -21573.961} C_VEL
LIN {X 0,Y 220.904,Z 728.73,A -85,B 0,C 180,E1 -21576.206,E2 -21576.206} C_VEL
LIN {X 0,Y 221.502,Z 727.006,A -85,B 0,C 180,E1 -21576.635,E2 -21576.635} C_VEL
LIN {X 0,Y 220.944,Z 721.163,A -85,B 0,C 180,E1 -21578.655,E2 -21578.655} C_VEL
LIN {X 0,Y 219.259,Z 713.492,A -85,B 0,C 180,E1 -21581.305,E2 -21581.305} C_VEL
LIN {X 0,Y 216.978,Z 706.309,A -85,B 0,C 180,E1 -21583.778,E2 -21583.778} C_VEL
LIN {X 0,Y 213.627,Z 698.267,A -85,B 0,C 180,E1 -21586.686,E2 -21586.686} C_VEL
LIN {X 0,Y 209.537,Z 690.308,A -85,B 0,C 180,E1 -21589.775,E2 -21589.775} C_VEL
LIN {X 0,Y 204.314,Z 682.089,A -85,B 0,C 180,E1 -21593.464,E2 -21593.464} C_VEL
LIN {X 0,Y 203.746,Z 680.936,A -85,B 0,C 180,E1 -21593.924,E2 -21593.924} C_VEL
LIN {X 0,Y 201.476,Z 679.025,A -85,B 0,C 180,E1 -21595.373,E2 -21595.373} C_VEL
LIN {X 0,Y 200.34,Z 676.83,A -85,B 0,C 180,E1 -21596.292,E2 -21596.292} C_VEL
LIN {X 0,Y 200.115,Z 675.543,A -85,B 0,C 180,E1 -21596.666,E2 -21596.666} C_VEL
LIN {X 0,Y 200.483,Z 675.5,A -85,B 0,C 180,E1 -21600,E2 -21600} C_VEL
LIN {X 0,Y 200.035,Z 675.557,A -85,B 0,C 180,E1 -21604.03,E2 -21604.03} C_VEL
LIN {X 0,Y 200.123,Z 675.548,A -85,B 0,C 180,E1 -21608.076,E2 -21608.076} C_VEL
LIN {X 0,Y 199.941,Z 675.643,A -85,B 0,C 180,E1 -21611.66,E2 -21611.66} C_VEL
LIN {X 0,Y 200.244,Z 677.391,A -85,B 0,C 180,E1 -21616.307,E2 -21616.307} C_VEL
LIN {X 0,Y 200.644,Z 679.449,A -85,B 0,C 180,E1 -21620.504,E2 -21620.504} C_VEL
LIN {X 0,Y 201.172,Z 682.029,A -85,B 0,C 180,E1 -21624.786,E2 -21624.786} C_VEL
LIN {X 0,Y 201.891,Z 685.461,A -85,B 0,C 180,E1 -21629.508,E2 -21629.508} C_VEL
LIN {X 0,Y 202.951,Z 690.079,A -85,B 0,C 180,E1 -21634.847,E2 -21634.847} C_VEL
LIN {X 0,Y 203.645,Z 693.618,A -85,B 0,C 180,E1 -21638.404,E2 -21638.404} C_VEL
LIN {X 0,Y 204.602,Z 698.811,A -85,B 0,C 180,E1 -21643.055,E2 -21643.055} C_VEL
LIN {X 0,Y 204.683,Z 699.199,A -85,B 0,C 180,E1 -21643.287,E2 -21643.287} C_VEL
LIN {X 0,Y 206.158,Z 703.024,A -85,B 0,C 180,E1 -21644.247,E2 -21644.247} C_VEL
LIN {X 0,Y 208.537,Z 706.861,A -85,B 0,C 180,E1 -21645.576,E2 -21645.576} C_VEL
LIN {X 0,Y 210.361,Z 711.325,A -85,B 0,C 180,E1 -21646.722,E2 -21646.722} C_VEL
LIN {X 0,Y 211.423,Z 713.595,A -85,B 0,C 180,E1 -21647.348,E2 -21647.348} C_VEL
LIN {X 0,Y 212.557,Z 717.883,A -85,B 0,C 180,E1 -21648.219,E2 -21648.219} C_VEL
LIN {X 0,Y 214.388,Z 730.212,A -85,B 0,C 180,E1 -21650.479,E2 -21650.479} C_VEL
LIN {X 0,Y 215.186,Z 743.333,A -85,B 0,C 180,E1 -21652.886,E2 -21652.886} C_VEL
LIN {X 0,Y 214.842,Z 755.144,A -85,B 0,C 180,E1 -21655.171,E2 -21655.171} C_VEL
LIN {X 0,Y 213.864,Z 759.976,A -85,B 0,C 180,E1 -21656.05,E2 -21656.05} C_VEL
LIN {X 0,Y 211.902,Z 764.771,A -85,B 0,C 180,E1 -21656.839,E2 -21656.839} C_VEL
LIN {X 0,Y 206.195,Z 775.41,A -85,B 0,C 180,E1 -21658.774,E2 -21658.774} C_VEL
LIN {X 0,Y 204.437,Z 779.65,A -85,B 0,C 180,E1 -21659.84,E2 -21659.84} C_VEL
LIN {X 0,Y 201.876,Z 788.221,A -85,B 0,C 180,E1 -21662.529,E2 -21662.529} C_VEL
LIN {X 0,Y 201.245,Z 790.699,A -85,B 0,C 180,E1 -21663.349,E2 -21663.349} C_VEL
LIN {X 0,Y 200.572,Z 796.184,A -85,B 0,C 180,E1 -21664.302,E2 -21664.302} C_VEL
LIN {X 0,Y 198.258,Z 807.111,A -85,B 0,C 180,E1 -21666.496,E2 -21666.496} C_VEL
LIN {X 0,Y 196.045,Z 816.875,A -85,B 0,C 180,E1 -21668.992,E2 -21668.992} C_VEL
LIN {X 0,Y 194.326,Z 824.944,A -85,B 0,C 180,E1 -21671.55,E2 -21671.55} C_VEL
LIN {X 0,Y 192.621,Z 832.842,A -85,B 0,C 180,E1 -21674.66,E2 -21674.66} C_VEL
LIN {X 0,Y 191.603,Z 838.175,A -85,B 0,C 180,E1 -21677.285,E2 -21677.285} C_VEL
LIN {X 0,Y 190.851,Z 843.366,A -85,B 0,C 180,E1 -21680.46,E2 -21680.46} C_VEL
LIN {X 0,Y 190.424,Z 847.338,A -85,B 0,C 180,E1 -21683.642,E2 -21683.642} C_VEL
LIN {X 0,Y 190.317,Z 849.355,A -85,B 0,C 180,E1 -21685.763,E2 -21685.763} C_VEL
LIN {X 0,Y 190.35,Z 850.941,A -85,B 0,C 180,E1 -21687.883,E2 -21687.883} C_VEL
LIN {X 0,Y 190.455,Z 852.109,A -85,B 0,C 180,E1 -21689.999,E2 -21689.999} C_VEL
LIN {X 0,Y 190.294,Z 852.808,A -85,B 0,C 180,E1 -21692.115,E2 -21692.115} C_VEL
LIN {X 0,Y 190.353,Z 853.015,A -85,B 0,C 180,E1 -21696.358,E2 -21696.358} C_VEL
LIN {X 0,Y 190.629,Z 852.548,A -85,B 0,C 180,E1 -21698.479,E2 -21698.479} C_VEL
LIN {X 0,Y 191.849,Z 850.382,A -85,B 0,C 180,E1 -21702.696,E2 -21702.696} C_VEL
LIN {X 0,Y 193.915,Z 846.64,A -85,B 0,C 180,E1 -21706.853,E2 -21706.853} C_VEL
LIN {X 0,Y 196.336,Z 842.685,A -85,B 0,C 180,E1 -21709.879,E2 -21709.879} C_VEL
LIN {X 0,Y 199.829,Z 836.474,A -85,B 0,C 180,E1 -21713.421,E2 -21713.421} C_VEL
LIN {X 0,Y 203.112,Z 830.209,A -85,B 0,C 180,E1 -21716.177,E2 -21716.177} C_VEL
LIN {X 0,Y 207.105,Z 822.281,A -85,B 0,C 180,E1 -21718.917,E2 -21718.917} C_VEL
LIN {X 0,Y 210.929,Z 814.311,A -85,B 0,C 180,E1 -21721.093,E2 -21721.093} C_VEL
LIN {X 0,Y 214.46,Z 805.797,A -85,B 0,C 180,E1 -21723.01,E2 -21723.01} C_VEL
LIN {X 0,Y 217.984,Z 794.479,A -85,B 0,C 180,E1 -21725.19,E2 -21725.19} C_VEL
LIN {X 0,Y 220.239,Z 784.833,A -85,B 0,C 180,E1 -21726.778,E2 -21726.778} C_VEL
LIN {X 0,Y 221.34,Z 773.886,A -85,B 0,C 180,E1 -21728.606,E2 -21728.606} C_VEL
LIN {X 0,Y 221.222,Z 763.701,A -85,B 0,C 180,E1 -21730.318,E2 -21730.318} C_VEL
LIN {X 0,Y 219.923,Z 752.181,A -85,B 0,C 180,E1 -21732.359,E2 -21732.359} C_VEL
LIN {X 0,Y 217.384,Z 740.392,A -85,B 0,C 180,E1 -21734.662,E2 -21734.662} C_VEL
LIN {X 0,Y 216.061,Z 736.515,A -85,B 0,C 180,E1 -21735.691,E2 -21735.691} C_VEL
LIN {X 0,Y 215.684,Z 731.658,A -85,B 0,C 180,E1 -21738.541,E2 -21738.541} C_VEL
LIN {X 0,Y 215.558,Z 727.146,A -85,B 0,C 180,E1 -21741.722,E2 -21741.722} C_VEL
LIN {X 0,Y 214.915,Z 724.357,A -85,B 0,C 180,E1 -21744.836,E2 -21744.836} C_VEL
LIN {X 0,Y 214.575,Z 723.533,A -85,B 0,C 180,E1 -21746.165,E2 -21746.165} C_VEL
LIN {X 0,Y 213.406,Z 722.175,A -85,B 0,C 180,E1 -21750.397,E2 -21750.397} C_VEL
LIN {X 0,Y 212.78,Z 721.947,A -85,B 0,C 180,E1 -21754.571,E2 -21754.571} C_VEL
LIN {X 0,Y 212.366,Z 722.875,A -85,B 0,C 180,E1 -21758.652,E2 -21758.652} C_VEL
LIN {X 0,Y 212.273,Z 724.705,A -85,B 0,C 180,E1 -21762.664,E2 -21762.664} C_VEL
LIN {X 0,Y 212.332,Z 727.37,A -85,B 0,C 180,E1 -21766.603,E2 -21766.603} C_VEL
LIN {X 0,Y 212.428,Z 730.847,A -85,B 0,C 180,E1 -21770.478,E2 -21770.478} C_VEL
LIN {X 0,Y 212.342,Z 734.317,A -85,B 0,C 180,E1 -21773.449,E2 -21773.449} C_VEL
LIN {X 0,Y 214.999,Z 739.95,A -85,B 0,C 180,E1 -21775.488,E2 -21775.488} C_VEL
LIN {X 0,Y 216.486,Z 744.82,A -85,B 0,C 180,E1 -21776.807,E2 -21776.807} C_VEL
LIN {X 0,Y 218.497,Z 754.078,A -85,B 0,C 180,E1 -21778.992,E2 -21778.992} C_VEL
LIN {X 0,Y 219.951,Z 764.994,A -85,B 0,C 180,E1 -21781.429,E2 -21781.429} C_VEL
LIN {X 0,Y 220.319,Z 775.342,A -85,B 0,C 180,E1 -21783.658,E2 -21783.658} C_VEL
LIN {X 0,Y 219.702,Z 784.966,A -85,B 0,C 180,E1 -21785.757,E2 -21785.757} C_VEL
LIN {X 0,Y 218.806,Z 790.392,A -85,B 0,C 180,E1 -21786.936,E2 -21786.936} C_VEL
LIN {X 0,Y 214.713,Z 800.728,A -85,B 0,C 180,E1 -21788.944,E2 -21788.944} C_VEL
LIN {X 0,Y 210.86,Z 809.309,A -85,B 0,C 180,E1 -21791.049,E2 -21791.049} C_VEL
LIN {X 0,Y 206.486,Z 818.013,A -85,B 0,C 180,E1 -21793.783,E2 -21793.783} C_VEL
LIN {X 0,Y 202.66,Z 825.074,A -85,B 0,C 180,E1 -21796.624,E2 -21796.624} C_VEL
LIN {X 0,Y 199.274,Z 830.854,A -85,B 0,C 180,E1 -21799.626,E2 -21799.626} C_VEL
LIN {X 0,Y 196.031,Z 835.97,A -85,B 0,C 180,E1 -21803.226,E2 -21803.226} C_VEL
LIN {X 0,Y 194.269,Z 838.601,A -85,B 0,C 180,E1 -21805.729,E2 -21805.729} C_VEL
LIN {X 0,Y 192.572,Z 840.951,A -85,B 0,C 180,E1 -21808.853,E2 -21808.853} C_VEL
LIN {X 0,Y 191.182,Z 842.48,A -85,B 0,C 180,E1 -21812.278,E2 -21812.278} C_VEL
LIN {X 0,Y 190.14,Z 842.925,A -85,B 0,C 180,E1 -21816.256,E2 -21816.256} C_VEL
LIN {X 0,Y 189.803,Z 842.428,A -85,B 0,C 180,E1 -21819.011,E2 -21819.011} C_VEL
LIN {X 0,Y 189.689,Z 841.012,A -85,B 0,C 180,E1 -21822.185,E2 -21822.185} C_VEL
LIN {X 0,Y 189.892,Z 838.713,A -85,B 0,C 180,E1 -21825.318,E2 -21825.318} C_VEL
LIN {X 0,Y 190.435,Z 835.533,A -85,B 0,C 180,E1 -21828.374,E2 -21828.374} C_VEL
LIN {X 0,Y 191.159,Z 831.507,A -85,B 0,C 180,E1 -21831.319,E2 -21831.319} C_VEL
LIN {X 0,Y 192.544,Z 825.221,A -85,B 0,C 180,E1 -21834.875,E2 -21834.875} C_VEL
LIN {X 0,Y 193.887,Z 818.925,A -85,B 0,C 180,E1 -21837.681,E2 -21837.681} C_VEL
LIN {X 0,Y 195.924,Z 810.263,A -85,B 0,C 180,E1 -21840.754,E2 -21840.754} C_VEL
LIN {X 0,Y 197.888,Z 801.478,A -85,B 0,C 180,E1 -21843.262,E2 -21843.262} C_VEL
LIN {X 0,Y 199.983,Z 791.967,A -85,B 0,C 180,E1 -21845.466,E2 -21845.466} C_VEL
LIN {X 0,Y 202.213,Z 780.781,A -85,B 0,C 180,E1 -21847.524,E2 -21847.524} C_VEL
LIN {X 0,Y 202.994,Z 774.609,A -85,B 0,C 180,E1 -21848.498,E2 -21848.498} C_VEL
LIN {X 0,Y 202.133,Z 763.467,A -85,B 0,C 180,E1 -21850.185,E2 -21850.185} C_VEL
LIN {X 0,Y 200.684,Z 750.614,A -85,B 0,C 180,E1 -21851.762,E2 -21851.762} C_VEL
LIN {X 0,Y 198.571,Z 736.842,A -85,B 0,C 180,E1 -21853.078,E2 -21853.078} C_VEL
LIN {X 0,Y 197.735,Z 732.115,A -85,B 0,C 180,E1 -21853.482,E2 -21853.482} C_VEL
LIN {X 0,Y 199.47,Z 720.836,A -85,B 0,C 180,E1 -21858.827,E2 -21858.827} C_VEL
LIN {X 0,Y 200.489,Z 714.287,A -85,B 0,C 180,E1 -21861.941,E2 -21861.941} C_VEL
LIN {X 0,Y 200.081,Z 708.476,A -85,B 0,C 180,E1 -21864.963,E2 -21864.963} C_VEL
LIN {X 0,Y 198.716,Z 699.271,A -85,B 0,C 180,E1 -21870.001,E2 -21870.001} C_VEL
LIN {X 0,Y 197.85,Z 694.624,A -85,B 0,C 180,E1 -21872.658,E2 -21872.658} C_VEL
LIN {X 0,Y 195.896,Z 687.01,A -85,B 0,C 180,E1 -21877.279,E2 -21877.279} C_VEL
LIN {X 0,Y 197.864,Z 689.458,A -85,B 0,C 180,E1 -21877.912,E2 -21877.912} C_VEL
LIN {X 0,Y 201.573,Z 701.247,A -85,B 0,C 180,E1 -21880.345,E2 -21880.345} C_VEL
LIN {X 0,Y 204.119,Z 711.399,A -85,B 0,C 180,E1 -21882.738,E2 -21882.738} C_VEL
LIN {X 0,Y 204.377,Z 712.804,A -85,B 0,C 180,E1 -21883.094,E2 -21883.094} C_VEL
LIN {X 0,Y 202.443,Z 722.132,A -85,B 0,C 180,E1 -21885.199,E2 -21885.199} C_VEL
LIN {X 0,Y 200.333,Z 731.597,A -85,B 0,C 180,E1 -21887.833,E2 -21887.833} C_VEL
LIN {X 0,Y 198.329,Z 739.954,A -85,B 0,C 180,E1 -21890.755,E2 -21890.755} C_VEL
LIN {X 0,Y 196.36,Z 747.973,A -85,B 0,C 180,E1 -21894.306,E2 -21894.306} C_VEL
LIN {X 0,Y 194.965,Z 754.184,A -85,B 0,C 180,E1 -21897.946,E2 -21897.946} C_VEL
LIN {X 0,Y 193.955,Z 758.954,A -85,B 0,C 180,E1 -21901.697,E2 -21901.697} C_VEL
LIN {X 0,Y 193.443,Z 762.328,A -85,B 0,C 180,E1 -21905.543,E2 -21905.543} C_VEL
LIN {X 0,Y 193.467,Z 763.799,A -85,B 0,C 180,E1 -21908.139,E2 -21908.139} C_VEL
LIN {X 0,Y 193.796,Z 764.669,A -85,B 0,C 180,E1 -21910.752,E2 -21910.752} C_VEL
LIN {X 0,Y 194.565,Z 764.923,A -85,B 0,C 180,E1 -21913.745,E2 -21913.745} C_VEL
LIN {X 0,Y 195.817,Z 764.258,A -85,B 0,C 180,E1 -21917.006,E2 -21917.006} C_VEL
LIN {X 0,Y 197.496,Z 762.64,A -85,B 0,C 180,E1 -21920.168,E2 -21920.168} C_VEL
LIN {X 0,Y 199.997,Z 759.346,A -85,B 0,C 180,E1 -21923.925,E2 -21923.925} C_VEL
LIN {X 0,Y 202.169,Z 756.089,A -85,B 0,C 180,E1 -21926.545,E2 -21926.545} C_VEL
LIN {X 0,Y 205.397,Z 750.706,A -85,B 0,C 180,E1 -21929.766,E2 -21929.766} C_VEL
LIN {X 0,Y 209.141,Z 743.669,A -85,B 0,C 180,E1 -21932.936,E2 -21932.936} C_VEL
LIN {X 0,Y 212.92,Z 735.417,A -85,B 0,C 180,E1 -21935.76,E2 -21935.76} C_VEL
LIN {X 0,Y 215.502,Z 729.249,A -85,B 0,C 180,E1 -21937.469,E2 -21937.469} C_VEL
LIN {X 0,Y 214.846,Z 722.712,A -85,B 0,C 180,E1 -21939.912,E2 -21939.912} C_VEL
LIN {X 0,Y 213.18,Z 715.072,A -85,B 0,C 180,E1 -21942.74,E2 -21942.74} C_VEL
LIN {X 0,Y 210.426,Z 706.494,A -85,B 0,C 180,E1 -21945.987,E2 -21945.987} C_VEL
LIN {X 0,Y 207.187,Z 699.172,A -85,B 0,C 180,E1 -21948.958,E2 -21948.958} C_VEL
LIN {X 0,Y 203.477,Z 692.178,A -85,B 0,C 180,E1 -21952.059,E2 -21952.059} C_VEL
LIN {X 0,Y 201.164,Z 688.293,A -85,B 0,C 180,E1 -21953.984,E2 -21953.984} C_VEL
LIN {X 0,Y 197.921,Z 684.035,A -85,B 0,C 180,E1 -21956.559,E2 -21956.559} C_VEL
LIN {X 0,Y 197.147,Z 681.912,A -85,B 0,C 180,E1 -21957.431,E2 -21957.431} C_VEL
LIN {X 0,Y 194.741,Z 679.781,A -85,B 0,C 180,E1 -21959.354,E2 -21959.354} C_VEL
LIN {X 0,Y 193.479,Z 677.069,A -85,B 0,C 180,E1 -21960.716,E2 -21960.716} C_VEL
LIN {X 0,Y 193.344,Z 676.386,A -85,B 0,C 180,E1 -21960.977,E2 -21960.977} C_VEL
LIN {X 0,Y 193.041,Z 676.755,A -85,B 0,C 180,E1 -21966.271,E2 -21966.271} C_VEL
LIN {X 0,Y 193.285,Z 677.717,A -85,B 0,C 180,E1 -21970.475,E2 -21970.475} C_VEL
LIN {X 0,Y 193.427,Z 679.192,A -85,B 0,C 180,E1 -21974.735,E2 -21974.735} C_VEL
LIN {X 0,Y 193.858,Z 681.33,A -85,B 0,C 180,E1 -21979.508,E2 -21979.508} C_VEL
LIN {X 0,Y 194.267,Z 683.548,A -85,B 0,C 180,E1 -21983.45,E2 -21983.45} C_VEL
LIN {X 0,Y 194.917,Z 686.564,A -85,B 0,C 180,E1 -21987.952,E2 -21987.952} C_VEL
LIN {X 0,Y 195.684,Z 690.244,A -85,B 0,C 180,E1 -21992.597,E2 -21992.597} C_VEL
LIN {X 0,Y 196.436,Z 693.446,A -85,B 0,C 180,E1 -21996.181,E2 -21996.181} C_VEL
LIN {X 0,Y 197.036,Z 696.63,A -85,B 0,C 180,E1 -21999.275,E2 -21999.275} C_VEL
LIN {X 0,Y 198.646,Z 700.622,A -85,B 0,C 180,E1 -22000.559,E2 -22000.559} C_VEL
LIN {X 0,Y 201.425,Z 705.12,A -85,B 0,C 180,E1 -22002.45,E2 -22002.45} C_VEL
LIN {X 0,Y 203.209,Z 709.453,A -85,B 0,C 180,E1 -22003.765,E2 -22003.765} C_VEL
LIN {X 0,Y 204.739,Z 712.205,A -85,B 0,C 180,E1 -22004.739,E2 -22004.739} C_VEL
LIN {X 0,Y 207.148,Z 718.412,A -85,B 0,C 180,E1 -22006.487,E2 -22006.487} C_VEL
LIN {X 0,Y 208.491,Z 726.501,A -85,B 0,C 180,E1 -22008.146,E2 -22008.146} C_VEL
LIN {X 0,Y 209.317,Z 736.056,A -85,B 0,C 180,E1 -22010.023,E2 -22010.023} C_VEL
LIN {X 0,Y 209.4,Z 748.68,A -85,B 0,C 180,E1 -22012.546,E2 -22012.546} C_VEL
LIN {X 0,Y 208.606,Z 758.949,A -85,B 0,C 180,E1 -22014.711,E2 -22014.711} C_VEL
LIN {X 0,Y 206.799,Z 770.281,A -85,B 0,C 180,E1 -22017.349,E2 -22017.349} C_VEL
LIN {X 0,Y 204.437,Z 779.65,A -85,B 0,C 180,E1 -22019.84,E2 -22019.84} C_VEL
LIN {X 0,Y 202.982,Z 782.543,A -85,B 0,C 180,E1 -22020.595,E2 -22020.595} C_VEL
LIN {X 0,Y 199.009,Z 787.019,A -85,B 0,C 180,E1 -22021.67,E2 -22021.67} C_VEL
LIN {X 0,Y 195.287,Z 790.96,A -85,B 0,C 180,E1 -22022.689,E2 -22022.689} C_VEL
LIN {X 0,Y 194.135,Z 793.86,A -85,B 0,C 180,E1 -22023.31,E2 -22023.31} C_VEL
LIN {X 0,Y 191.893,Z 804.317,A -85,B 0,C 180,E1 -22025.379,E2 -22025.379} C_VEL
LIN {X 0,Y 189.683,Z 814.579,A -85,B 0,C 180,E1 -22027.943,E2 -22027.943} C_VEL
LIN {X 0,Y 187.568,Z 823.802,A -85,B 0,C 180,E1 -22030.86,E2 -22030.86} C_VEL
LIN {X 0,Y 185.744,Z 831.863,A -85,B 0,C 180,E1 -22034.078,E2 -22034.078} C_VEL
LIN {X 0,Y 184.655,Z 837.333,A -85,B 0,C 180,E1 -22036.798,E2 -22036.798} C_VEL
LIN {X 0,Y 183.809,Z 842.653,A -85,B 0,C 180,E1 -22040.091,E2 -22040.091} C_VEL
LIN {X 0,Y 183.367,Z 846.745,A -85,B 0,C 180,E1 -22043.396,E2 -22043.396} C_VEL
LIN {X 0,Y 183.228,Z 848.996,A -85,B 0,C 180,E1 -22045.774,E2 -22045.774} C_VEL
LIN {X 0,Y 183.253,Z 850.493,A -85,B 0,C 180,E1 -22047.801,E2 -22047.801} C_VEL
LIN {X 0,Y 183.37,Z 851.714,A -85,B 0,C 180,E1 -22049.999,E2 -22049.999} C_VEL
LIN {X 0,Y 183.14,Z 852.821,A -85,B 0,C 180,E1 -22053.839,E2 -22053.839} C_VEL
LIN {X 0,Y 183.294,Z 852.838,A -85,B 0,C 180,E1 -22056.604,E2 -22056.604} C_VEL
LIN {X 0,Y 184.139,Z 851.64,A -85,B 0,C 180,E1 -22061,E2 -22061} C_VEL
LIN {X 0,Y 185.855,Z 848.839,A -85,B 0,C 180,E1 -22065.348,E2 -22065.348} C_VEL
LIN {X 0,Y 187.932,Z 845.683,A -85,B 0,C 180,E1 -22068.533,E2 -22068.533} C_VEL
LIN {X 0,Y 190.703,Z 841.516,A -85,B 0,C 180,E1 -22071.624,E2 -22071.624} C_VEL
LIN {X 0,Y 193.766,Z 836.116,A -85,B 0,C 180,E1 -22074.737,E2 -22074.737} C_VEL
LIN {X 0,Y 198.184,Z 828.597,A -85,B 0,C 180,E1 -22078.024,E2 -22078.024} C_VEL
LIN {X 0,Y 201.689,Z 821.886,A -85,B 0,C 180,E1 -22080.347,E2 -22080.347} C_VEL
LIN {X 0,Y 205.825,Z 813.86,A -85,B 0,C 180,E1 -22082.532,E2 -22082.532} C_VEL
LIN {X 0,Y 209.421,Z 805.334,A -85,B 0,C 180,E1 -22084.492,E2 -22084.492} C_VEL
LIN {X 0,Y 213.213,Z 794.015,A -85,B 0,C 180,E1 -22086.7,E2 -22086.7} C_VEL
LIN {X 0,Y 215.435,Z 784.774,A -85,B 0,C 180,E1 -22088.302,E2 -22088.302} C_VEL
LIN {X 0,Y 216.526,Z 774.304,A -85,B 0,C 180,E1 -22090.151,E2 -22090.151} C_VEL
LIN {X 0,Y 216.59,Z 764.338,A -85,B 0,C 180,E1 -22091.952,E2 -22091.952} C_VEL
LIN {X 0,Y 215.615,Z 753.847,A -85,B 0,C 180,E1 -22093.947,E2 -22093.947} C_VEL
LIN {X 0,Y 213.683,Z 743.45,A -85,B 0,C 180,E1 -22096.164,E2 -22096.164} C_VEL
LIN {X 0,Y 212.075,Z 740.076,A -85,B 0,C 180,E1 -22097.381,E2 -22097.381} C_VEL
LIN {X 0,Y 210.397,Z 736.238,A -85,B 0,C 180,E1 -22098.881,E2 -22098.881} C_VEL
LIN {X 0,Y 210.309,Z 732.676,A -85,B 0,C 180,E1 -22101.381,E2 -22101.381} C_VEL
LIN {X 0,Y 210.057,Z 730.44,A -85,B 0,C 180,E1 -22103.413,E2 -22103.413} C_VEL
LIN {X 0,Y 209.669,Z 728.992,A -85,B 0,C 180,E1 -22105.261,E2 -22105.261} C_VEL
LIN {X 0,Y 208.966,Z 727.918,A -85,B 0,C 180,E1 -22107.444,E2 -22107.444} C_VEL
LIN {X 0,Y 207.919,Z 726.797,A -85,B 0,C 180,E1 -22111.756,E2 -22111.756} C_VEL
LIN {X 0,Y 207.586,Z 726.653,A -85,B 0,C 180,E1 -22113.888,E2 -22113.888} C_VEL
LIN {X 0,Y 207.018,Z 727.361,A -85,B 0,C 180,E1 -22118.072,E2 -22118.072} C_VEL
LIN {X 0,Y 206.79,Z 729.005,A -85,B 0,C 180,E1 -22122.189,E2 -22122.189} C_VEL
LIN {X 0,Y 206.714,Z 731.512,A -85,B 0,C 180,E1 -22126.232,E2 -22126.232} C_VEL
LIN {X 0,Y 206.782,Z 734.692,A -85,B 0,C 180,E1 -22129.842,E2 -22129.842} C_VEL
LIN {X 0,Y 208.95,Z 739.118,A -85,B 0,C 180,E1 -22131.964,E2 -22131.964} C_VEL
LIN {X 0,Y 209.994,Z 740.903,A -85,B 0,C 180,E1 -22132.872,E2 -22132.872} C_VEL
LIN {X 0,Y 211.911,Z 745.522,A -85,B 0,C 180,E1 -22134.626,E2 -22134.626} C_VEL
LIN {X 0,Y 213.373,Z 751.744,A -85,B 0,C 180,E1 -22136.353,E2 -22136.353} C_VEL
LIN {X 0,Y 214.776,Z 762.24,A -85,B 0,C 180,E1 -22138.891,E2 -22138.891} C_VEL
LIN {X 0,Y 215.338,Z 771.408,A -85,B 0,C 180,E1 -22141.05,E2 -22141.05} C_VEL
LIN {X 0,Y 214.957,Z 782.156,A -85,B 0,C 180,E1 -22143.514,E2 -22143.514} C_VEL
LIN {X 0,Y 213.558,Z 791.43,A -85,B 0,C 180,E1 -22145.666,E2 -22145.666} C_VEL
LIN {X 0,Y 209.31,Z 801.612,A -85,B 0,C 180,E1 -22147.718,E2 -22147.718} C_VEL
LIN {X 0,Y 205.271,Z 810.084,A -85,B 0,C 180,E1 -22149.857,E2 -22149.857} C_VEL
LIN {X 0,Y 200.651,Z 818.706,A -85,B 0,C 180,E1 -22152.644,E2 -22152.644} C_VEL
LIN {X 0,Y 196.797,Z 825.292,A -85,B 0,C 180,E1 -22155.379,E2 -22155.379} C_VEL
LIN {X 0,Y 192.909,Z 831.46,A -85,B 0,C 180,E1 -22158.703,E2 -22158.703} C_VEL
LIN {X 0,Y 189.685,Z 836.166,A -85,B 0,C 180,E1 -22162.143,E2 -22162.143} C_VEL
LIN {X 0,Y 187.121,Z 839.577,A -85,B 0,C 180,E1 -22165.66,E2 -22165.66} C_VEL
LIN {X 0,Y 185.092,Z 841.981,A -85,B 0,C 180,E1 -22169.578,E2 -22169.578} C_VEL
LIN {X 0,Y 183.889,Z 842.961,A -85,B 0,C 180,E1 -22172.777,E2 -22172.777} C_VEL
LIN {X 0,Y 183.036,Z 843.083,A -85,B 0,C 180,E1 -22176.263,E2 -22176.263} C_VEL
LIN {X 0,Y 182.643,Z 842.239,A -85,B 0,C 180,E1 -22179.685,E2 -22179.685} C_VEL
LIN {X 0,Y 182.667,Z 839.942,A -85,B 0,C 180,E1 -22183.831,E2 -22183.831} C_VEL
LIN {X 0,Y 183.284,Z 835.931,A -85,B 0,C 180,E1 -22188.115,E2 -22188.115} C_VEL
LIN {X 0,Y 184.017,Z 831.966,A -85,B 0,C 180,E1 -22191.179,E2 -22191.179} C_VEL
LIN {X 0,Y 185.351,Z 825.858,A -85,B 0,C 180,E1 -22194.819,E2 -22194.819} C_VEL
LIN {X 0,Y 186.748,Z 819.617,A -85,B 0,C 180,E1 -22197.754,E2 -22197.754} C_VEL
LIN {X 0,Y 188.6,Z 811.934,A -85,B 0,C 180,E1 -22200.668,E2 -22200.668} C_VEL
LIN {X 0,Y 190.794,Z 802.557,A -85,B 0,C 180,E1 -22203.506,E2 -22203.506} C_VEL
LIN {X 0,Y 193.211,Z 791.884,A -85,B 0,C 180,E1 -22206.082,E2 -22206.082} C_VEL
LIN {X 0,Y 195.402,Z 781.293,A -85,B 0,C 180,E1 -22208.092,E2 -22208.092} C_VEL
LIN {X 0,Y 196.191,Z 775.69,A -85,B 0,C 180,E1 -22209.01,E2 -22209.01} C_VEL
LIN {X 0,Y 195.387,Z 764.168,A -85,B 0,C 180,E1 -22210.84,E2 -22210.84} C_VEL
LIN {X 0,Y 194.031,Z 751.681,A -85,B 0,C 180,E1 -22212.461,E2 -22212.461} C_VEL
LIN {X 0,Y 191.947,Z 737.476,A -85,B 0,C 180,E1 -22213.87,E2 -22213.87} C_VEL
LIN {X 0,Y 190.967,Z 732.26,A -85,B 0,C 180,E1 -22214.344,E2 -22214.344} C_VEL
LIN {X 0,Y 192.822,Z 721.077,A -85,B 0,C 180,E1 -22219.768,E2 -22219.768} C_VEL
LIN {X 0,Y 193.65,Z 716.116,A -85,B 0,C 180,E1 -22222.179,E2 -22222.179} C_VEL
LIN {X 0,Y 193.41,Z 711.203,A -85,B 0,C 180,E1 -22224.789,E2 -22224.789} C_VEL
LIN {X 0,Y 192.078,Z 701.901,A -85,B 0,C 180,E1 -22230.001,E2 -22230.001} C_VEL
LIN {X 0,Y 191.269,Z 697.232,A -85,B 0,C 180,E1 -22232.727,E2 -22232.727} C_VEL
LIN {X 0,Y 189.569,Z 690.73,A -85,B 0,C 180,E1 -22236.868,E2 -22236.868} C_VEL
LIN {X 0,Y 192.245,Z 694.257,A -85,B 0,C 180,E1 -22237.827,E2 -22237.827} C_VEL
LIN {X 0,Y 195.54,Z 705.478,A -85,B 0,C 180,E1 -22240.354,E2 -22240.354} C_VEL
LIN {X 0,Y 197.592,Z 714.354,A -85,B 0,C 180,E1 -22242.584,E2 -22242.584} C_VEL
LIN {X 0,Y 195.259,Z 725.019,A -85,B 0,C 180,E1 -22245.128,E2 -22245.128} C_VEL
LIN {X 0,Y 193.051,Z 734.19,A -85,B 0,C 180,E1 -22247.89,E2 -22247.89} C_VEL
LIN {X 0,Y 190.99,Z 742.523,A -85,B 0,C 180,E1 -22251.026,E2 -22251.026} C_VEL
LIN {X 0,Y 189.364,Z 749.04,A -85,B 0,C 180,E1 -22254.096,E2 -22254.096} C_VEL
LIN {X 0,Y 187.911,Z 755.25,A -85,B 0,C 180,E1 -22257.874,E2 -22257.874} C_VEL
LIN {X 0,Y 186.87,Z 760.033,A -85,B 0,C 180,E1 -22261.772,E2 -22261.772} C_VEL
LIN {X 0,Y 186.469,Z 762.421,A -85,B 0,C 180,E1 -22264.428,E2 -22264.428} C_VEL
LIN {X 0,Y 186.405,Z 764.491,A -85,B 0,C 180,E1 -22267.65,E2 -22267.65} C_VEL
LIN {X 0,Y 186.845,Z 765.746,A -85,B 0,C 180,E1 -22271.212,E2 -22271.212} C_VEL
LIN {X 0,Y 188.039,Z 765.88,A -85,B 0,C 180,E1 -22275.247,E2 -22275.247} C_VEL
LIN {X 0,Y 189.237,Z 765.161,A -85,B 0,C 180,E1 -22278.049,E2 -22278.049} C_VEL
LIN {X 0,Y 191.124,Z 763.427,A -85,B 0,C 180,E1 -22281.309,E2 -22281.309} C_VEL
LIN {X 0,Y 193.28,Z 760.814,A -85,B 0,C 180,E1 -22284.424,E2 -22284.424} C_VEL
LIN {X 0,Y 196.378,Z 756.426,A -85,B 0,C 180,E1 -22288.003,E2 -22288.003} C_VEL
LIN {X 0,Y 200.045,Z 750.568,A -85,B 0,C 180,E1 -22291.439,E2 -22291.439} C_VEL
LIN {X 0,Y 204.072,Z 743.187,A -85,B 0,C 180,E1 -22294.633,E2 -22294.633} C_VEL
LIN {X 0,Y 208.193,Z 734.664,A -85,B 0,C 180,E1 -22297.472,E2 -22297.472} C_VEL
LIN {X 0,Y 209.465,Z 731.599,A -85,B 0,C 180,E1 -22298.342,E2 -22298.342} C_VEL
LIN {X 0,Y 208.927,Z 725.333,A -85,B 0,C 180,E1 -22300.854,E2 -22300.854} C_VEL
LIN {X 0,Y 207.6,Z 718.358,A -85,B 0,C 180,E1 -22303.643,E2 -22303.643} C_VEL
LIN {X 0,Y 205.342,Z 710.704,A -85,B 0,C 180,E1 -22306.77,E2 -22306.77} C_VEL
LIN {X 0,Y 202.397,Z 703.408,A -85,B 0,C 180,E1 -22310.002,E2 -22310.002} C_VEL
LIN {X 0,Y 199.453,Z 697.353,A -85,B 0,C 180,E1 -22312.916,E2 -22312.916} C_VEL
LIN {X 0,Y 197.643,Z 694.034,A -85,B 0,C 180,E1 -22314.664,E2 -22314.664} C_VEL
LIN {X 0,Y 195.158,Z 690.628,A -85,B 0,C 180,E1 -22316.924,E2 -22316.924} C_VEL
LIN {X 0,Y 194.367,Z 688.502,A -85,B 0,C 180,E1 -22317.928,E2 -22317.928} C_VEL
LIN {X 0,Y 191.891,Z 685.509,A -85,B 0,C 180,E1 -22320.328,E2 -22320.328} C_VEL
LIN {X 0,Y 190.994,Z 683.142,A -85,B 0,C 180,E1 -22321.582,E2 -22321.582} C_VEL
LIN {X 0,Y 187.515,Z 681.105,A -85,B 0,C 180,E1 -22325.377,E2 -22325.377} C_VEL
LIN {X 0,Y 186.426,Z 679.38,A -85,B 0,C 180,E1 -22327.174,E2 -22327.174} C_VEL
LIN {X 0,Y 186.592,Z 680.566,A -85,B 0,C 180,E1 -22331.676,E2 -22331.676} C_VEL
LIN {X 0,Y 186.794,Z 681.842,A -85,B 0,C 180,E1 -22335.271,E2 -22335.271} C_VEL
LIN {X 0,Y 187.221,Z 684.101,A -85,B 0,C 180,E1 -22340.203,E2 -22340.203} C_VEL
LIN {X 0,Y 187.669,Z 686.445,A -85,B 0,C 180,E1 -22344.327,E2 -22344.327} C_VEL
LIN {X 0,Y 188.326,Z 689.622,A -85,B 0,C 180,E1 -22349.022,E2 -22349.022} C_VEL
LIN {X 0,Y 189.164,Z 693.342,A -85,B 0,C 180,E1 -22353.55,E2 -22353.55} C_VEL
LIN {X 0,Y 191.68,Z 698.936,A -85,B 0,C 180,E1 -22356.276,E2 -22356.276} C_VEL
LIN {X 0,Y 194.174,Z 702.654,A -85,B 0,C 180,E1 -22358.406,E2 -22358.406} C_VEL
LIN {X 0,Y 196.091,Z 707.397,A -85,B 0,C 180,E1 -22360.176,E2 -22360.176} C_VEL
LIN {X 0,Y 197.941,Z 710.641,A -85,B 0,C 180,E1 -22361.585,E2 -22361.585} C_VEL
LIN {X 0,Y 199.614,Z 714.973,A -85,B 0,C 180,E1 -22363.033,E2 -22363.033} C_VEL
LIN {X 0,Y 200.843,Z 717.656,A -85,B 0,C 180,E1 -22363.983,E2 -22363.983} C_VEL
LIN {X 0,Y 202.771,Z 723.148,A -85,B 0,C 180,E1 -22365.634,E2 -22365.634} C_VEL
LIN {X 0,Y 203.754,Z 732.338,A -85,B 0,C 180,E1 -22367.632,E2 -22367.632} C_VEL
LIN {X 0,Y 203.964,Z 744.187,A -85,B 0,C 180,E1 -22370.119,E2 -22370.119} C_VEL
LIN {X 0,Y 203.289,Z 754.669,A -85,B 0,C 180,E1 -22372.409,E2 -22372.409} C_VEL
LIN {X 0,Y 201.768,Z 765.325,A -85,B 0,C 180,E1 -22374.918,E2 -22374.918} C_VEL
LIN {X 0,Y 199.496,Z 775.373,A -85,B 0,C 180,E1 -22377.563,E2 -22377.563} C_VEL
LIN {X 0,Y 196.415,Z 785.065,A -85,B 0,C 180,E1 -22380.527,E2 -22380.527} C_VEL
LIN {X 0,Y 194.374,Z 791.625,A -85,B 0,C 180,E1 -22382.911,E2 -22382.911} C_VEL
LIN {X 0,Y 194.135,Z 793.86,A -85,B 0,C 180,E1 -22383.31,E2 -22383.31} C_VEL
LIN {X 0,Y 192.989,Z 797.183,A -85,B 0,C 180,E1 -22383.874,E2 -22383.874} C_VEL
LIN {X 0,Y 189.191,Z 802.164,A -85,B 0,C 180,E1 -22384.65,E2 -22384.65} C_VEL
LIN {X 0,Y 185.234,Z 806.909,A -85,B 0,C 180,E1 -22385.512,E2 -22385.512} C_VEL
LIN {X 0,Y 183.85,Z 809.864,A -85,B 0,C 180,E1 -22386.215,E2 -22386.215} C_VEL
LIN {X 0,Y 181.584,Z 819.535,A -85,B 0,C 180,E1 -22389.067,E2 -22389.067} C_VEL
LIN {X 0,Y 179.513,Z 828.283,A -85,B 0,C 180,E1 -22392.336,E2 -22392.336} C_VEL
LIN {X 0,Y 177.873,Z 835.409,A -85,B 0,C 180,E1 -22395.702,E2 -22395.702} C_VEL
LIN {X 0,Y 177.026,Z 840.215,A -85,B 0,C 180,E1 -22398.55,E2 -22398.55} C_VEL
LIN {X 0,Y 176.429,Z 844.843,A -85,B 0,C 180,E1 -22401.984,E2 -22401.984} C_VEL
LIN {X 0,Y 176.144,Z 848.73,A -85,B 0,C 180,E1 -22405.935,E2 -22405.935} C_VEL
LIN {X 0,Y 176.287,Z 851.312,A -85,B 0,C 180,E1 -22409.999,E2 -22409.999} C_VEL
LIN {X 0,Y 176.048,Z 852.461,A -85,B 0,C 180,E1 -22413.597,E2 -22413.597} C_VEL
LIN {X 0,Y 176.231,Z 852.661,A -85,B 0,C 180,E1 -22416.87,E2 -22416.87} C_VEL
LIN {X 0,Y 177.163,Z 851.591,A -85,B 0,C 180,E1 -22421.439,E2 -22421.439} C_VEL
LIN {X 0,Y 177.967,Z 850.495,A -85,B 0,C 180,E1 -22423.705,E2 -22423.705} C_VEL
LIN {X 0,Y 178.989,Z 848.979,A -85,B 0,C 180,E1 -22425.952,E2 -22425.952} C_VEL
LIN {X 0,Y 182.096,Z 844.716,A -85,B 0,C 180,E1 -22430.324,E2 -22430.324} C_VEL
LIN {X 0,Y 185.196,Z 840.37,A -85,B 0,C 180,E1 -22433.481,E2 -22433.481} C_VEL
LIN {X 0,Y 188.518,Z 834.942,A -85,B 0,C 180,E1 -22436.573,E2 -22436.573} C_VEL
LIN {X 0,Y 192.685,Z 828.23,A -85,B 0,C 180,E1 -22439.497,E2 -22439.497} C_VEL
LIN {X 0,Y 197.345,Z 819.981,A -85,B 0,C 180,E1 -22442.288,E2 -22442.288} C_VEL
LIN {X 0,Y 202.591,Z 809.869,A -85,B 0,C 180,E1 -22444.916,E2 -22444.916} C_VEL
LIN {X 0,Y 206.574,Z 799.711,A -85,B 0,C 180,E1 -22447.147,E2 -22447.147} C_VEL
LIN {X 0,Y 210.006,Z 788.493,A -85,B 0,C 180,E1 -22449.21,E2 -22449.21} C_VEL
LIN {X 0,Y 211.743,Z 777.612,A -85,B 0,C 180,E1 -22451.251,E2 -22451.251} C_VEL
LIN {X 0,Y 212.215,Z 767.216,A -85,B 0,C 180,E1 -22453.232,E2 -22453.232} C_VEL
LIN {X 0,Y 211.574,Z 756.085,A -85,B 0,C 180,E1 -22455.521,E2 -22455.521} C_VEL
LIN {X 0,Y 210.394,Z 748.125,A -85,B 0,C 180,E1 -22457.323,E2 -22457.323} C_VEL
LIN {X 0,Y 207.389,Z 741.333,A -85,B 0,C 180,E1 -22460.123,E2 -22460.123} C_VEL
LIN {X 0,Y 204.983,Z 735.881,A -85,B 0,C 180,E1 -22462.928,E2 -22462.928} C_VEL
LIN {X 0,Y 204.409,Z 733.715,A -85,B 0,C 180,E1 -22465.603,E2 -22465.603} C_VEL
LIN {X 0,Y 203.112,Z 731.977,A -85,B 0,C 180,E1 -22469.884,E2 -22469.884} C_VEL
LIN {X 0,Y 202.419,Z 731.472,A -85,B 0,C 180,E1 -22473.169,E2 -22473.169} C_VEL
LIN {X 0,Y 201.729,Z 731.897,A -85,B 0,C 180,E1 -22477.466,E2 -22477.466} C_VEL
LIN {X 0,Y 201.329,Z 733.362,A -85,B 0,C 180,E1 -22481.689,E2 -22481.689} C_VEL
LIN {X 0,Y 201.247,Z 734.965,A -85,B 0,C 180,E1 -22484.557,E2 -22484.557} C_VEL
LIN {X 0,Y 204.751,Z 741.337,A -85,B 0,C 180,E1 -22489.305,E2 -22489.305} C_VEL
LIN {X 0,Y 206.542,Z 745.399,A -85,B 0,C 180,E1 -22491.353,E2 -22491.353} C_VEL
LIN {X 0,Y 207.353,Z 747.116,A -85,B 0,C 180,E1 -22492.208,E2 -22492.208} C_VEL
LIN {X 0,Y 208.688,Z 751.117,A -85,B 0,C 180,E1 -22493.77,E2 -22493.77} C_VEL
LIN {X 0,Y 209.489,Z 755.473,A -85,B 0,C 180,E1 -22495.043,E2 -22495.043} C_VEL
LIN {X 0,Y 210.412,Z 765.667,A -85,B 0,C 180,E1 -22497.688,E2 -22497.688} C_VEL
LIN {X 0,Y 210.582,Z 774.954,A -85,B 0,C 180,E1 -22500,E2 -22500} C_VEL
LIN {X 0,Y 209.811,Z 784.74,A -85,B 0,C 180,E1 -22502.399,E2 -22502.399} C_VEL
LIN {X 0,Y 208.2,Z 793.323,A -85,B 0,C 180,E1 -22504.488,E2 -22504.488} C_VEL
LIN {X 0,Y 203.503,Z 803.687,A -85,B 0,C 180,E1 -22506.692,E2 -22506.692} C_VEL
LIN {X 0,Y 199.184,Z 811.96,A -85,B 0,C 180,E1 -22508.914,E2 -22508.914} C_VEL
LIN {X 0,Y 194.345,Z 820.37,A -85,B 0,C 180,E1 -22511.806,E2 -22511.806} C_VEL
LIN {X 0,Y 189.774,Z 827.488,A -85,B 0,C 180,E1 -22515.024,E2 -22515.024} C_VEL
LIN {X 0,Y 185.522,Z 833.579,A -85,B 0,C 180,E1 -22518.733,E2 -22518.733} C_VEL
LIN {X 0,Y 181.966,Z 838.168,A -85,B 0,C 180,E1 -22522.72,E2 -22522.72} C_VEL
LIN {X 0,Y 179.772,Z 840.748,A -85,B 0,C 180,E1 -22525.956,E2 -22525.956} C_VEL
LIN {X 0,Y 177.918,Z 842.58,A -85,B 0,C 180,E1 -22529.657,E2 -22529.657} C_VEL
LIN {X 0,Y 176.443,Z 843.367,A -85,B 0,C 180,E1 -22533.893,E2 -22533.893} C_VEL
LIN {X 0,Y 175.815,Z 843.113,A -85,B 0,C 180,E1 -22536.922,E2 -22536.922} C_VEL
LIN {X 0,Y 175.493,Z 841.947,A -85,B 0,C 180,E1 -22540.459,E2 -22540.459} C_VEL
LIN {X 0,Y 175.571,Z 839.885,A -85,B 0,C 180,E1 -22543.904,E2 -22543.904} C_VEL
LIN {X 0,Y 176.19,Z 835.982,A -85,B 0,C 180,E1 -22548.135,E2 -22548.135} C_VEL
LIN {X 0,Y 177.018,Z 831.634,A -85,B 0,C 180,E1 -22551.556,E2 -22551.556} C_VEL
LIN {X 0,Y 178.17,Z 826.441,A -85,B 0,C 180,E1 -22554.752,E2 -22554.752} C_VEL
LIN {X 0,Y 179.684,Z 819.964,A -85,B 0,C 180,E1 -22557.946,E2 -22557.946} C_VEL
LIN {X 0,Y 181.639,Z 812.072,A -85,B 0,C 180,E1 -22561.064,E2 -22561.064} C_VEL
LIN {X 0,Y 183.818,Z 803.01,A -85,B 0,C 180,E1 -22563.918,E2 -22563.918} C_VEL
LIN {X 0,Y 186.414,Z 791.98,A -85,B 0,C 180,E1 -22566.682,E2 -22566.682} C_VEL
LIN {X 0,Y 188.756,Z 780.974,A -85,B 0,C 180,E1 -22568.829,E2 -22568.829} C_VEL
LIN {X 0,Y 189.38,Z 776.189,A -85,B 0,C 180,E1 -22569.647,E2 -22569.647} C_VEL
LIN {X 0,Y 188.569,Z 763.568,A -85,B 0,C 180,E1 -22571.71,E2 -22571.71} C_VEL
LIN {X 0,Y 187.095,Z 750.369,A -85,B 0,C 180,E1 -22573.44,E2 -22573.44} C_VEL
LIN {X 0,Y 185.115,Z 737.107,A -85,B 0,C 180,E1 -22574.801,E2 -22574.801} C_VEL
LIN {X 0,Y 184.233,Z 732.433,A -85,B 0,C 180,E1 -22575.221,E2 -22575.221} C_VEL
LIN {X 0,Y 185.971,Z 722.764,A -85,B 0,C 180,E1 -22580.033,E2 -22580.033} C_VEL
LIN {X 0,Y 186.887,Z 716.914,A -85,B 0,C 180,E1 -22582.981,E2 -22582.981} C_VEL
LIN {X 0,Y 186.481,Z 712.032,A -85,B 0,C 180,E1 -22585.678,E2 -22585.678} C_VEL
LIN {X 0,Y 185.213,Z 702.682,A -85,B 0,C 180,E1 -22591.088,E2 -22591.088} C_VEL
LIN {X 0,Y 183.917,Z 697.365,A -85,B 0,C 180,E1 -22594.384,E2 -22594.384} C_VEL
LIN {X 0,Y 183.192,Z 694.291,A -85,B 0,C 180,E1 -22596.423,E2 -22596.423} C_VEL
LIN {X 0,Y 185.742,Z 697.261,A -85,B 0,C 180,E1 -22597.344,E2 -22597.344} C_VEL
LIN {X 0,Y 187.218,Z 701.393,A -85,B 0,C 180,E1 -22598.338,E2 -22598.338} C_VEL
LIN {X 0,Y 189.717,Z 710.763,A -85,B 0,C 180,E1 -22600.675,E2 -22600.675} C_VEL
LIN {X 0,Y 190.785,Z 715.515,A -85,B 0,C 180,E1 -22601.96,E2 -22601.96} C_VEL
LIN {X 0,Y 188.628,Z 725.325,A -85,B 0,C 180,E1 -22604.37,E2 -22604.37} C_VEL
LIN {X 0,Y 186.534,Z 733.932,A -85,B 0,C 180,E1 -22606.978,E2 -22606.978} C_VEL
LIN {X 0,Y 184.416,Z 742.116,A -85,B 0,C 180,E1 -22610.06,E2 -22610.06} C_VEL
LIN {X 0,Y 182.362,Z 750.1,A -85,B 0,C 180,E1 -22613.869,E2 -22613.869} C_VEL
LIN {X 0,Y 180.844,Z 756.323,A -85,B 0,C 180,E1 -22617.799,E2 -22617.799} C_VEL
LIN {X 0,Y 179.795,Z 761.17,A -85,B 0,C 180,E1 -22621.911,E2 -22621.911} C_VEL
LIN {X 0,Y 179.358,Z 764.466,A -85,B 0,C 180,E1 -22625.999,E2 -22625.999} C_VEL
LIN {X 0,Y 179.463,Z 765.939,A -85,B 0,C 180,E1 -22628.799,E2 -22628.799} C_VEL
LIN {X 0,Y 180.019,Z 766.892,A -85,B 0,C 180,E1 -22632.118,E2 -22632.118} C_VEL
LIN {X 0,Y 181.155,Z 766.969,A -85,B 0,C 180,E1 -22635.708,E2 -22635.708} C_VEL
LIN {X 0,Y 183.274,Z 765.691,A -85,B 0,C 180,E1 -22640.081,E2 -22640.081} C_VEL
LIN {X 0,Y 186.065,Z 762.846,A -85,B 0,C 180,E1 -22644.302,E2 -22644.302} C_VEL
LIN {X 0,Y 189.638,Z 758.28,A -85,B 0,C 180,E1 -22648.473,E2 -22648.473} C_VEL
LIN {X 0,Y 193.205,Z 753.082,A -85,B 0,C 180,E1 -22651.778,E2 -22651.778} C_VEL
LIN {X 0,Y 196.748,Z 747.244,A -85,B 0,C 180,E1 -22654.618,E2 -22654.618} C_VEL
LIN {X 0,Y 200.898,Z 739.514,A -85,B 0,C 180,E1 -22657.547,E2 -22657.547} C_VEL
LIN {X 0,Y 203.221,Z 734.688,A -85,B 0,C 180,E1 -22659.028,E2 -22659.028} C_VEL
LIN {X 0,Y 203.431,Z 731.732,A -85,B 0,C 180,E1 -22660.226,E2 -22660.226} C_VEL
LIN {X 0,Y 202.594,Z 724.488,A -85,B 0,C 180,E1 -22663.37,E2 -22663.37} C_VEL
LIN {X 0,Y 201.084,Z 717.638,A -85,B 0,C 180,E1 -22666.355,E2 -22666.355} C_VEL
LIN {X 0,Y 198.662,Z 710.165,A -85,B 0,C 180,E1 -22669.812,E2 -22669.812} C_VEL
LIN {X 0,Y 196.184,Z 704.287,A -85,B 0,C 180,E1 -22672.797,E2 -22672.797} C_VEL
LIN {X 0,Y 193.496,Z 699.016,A -85,B 0,C 180,E1 -22675.835,E2 -22675.835} C_VEL
LIN {X 0,Y 190.642,Z 693.928,A -85,B 0,C 180,E1 -22679.208,E2 -22679.208} C_VEL
LIN {X 0,Y 189.095,Z 691.449,A -85,B 0,C 180,E1 -22681.132,E2 -22681.132} C_VEL
LIN {X 0,Y 188.521,Z 689.709,A -85,B 0,C 180,E1 -22682.137,E2 -22682.137} C_VEL
LIN {X 0,Y 185.604,Z 687.863,A -85,B 0,C 180,E1 -22685.705,E2 -22685.705} C_VEL
LIN {X 0,Y 184.664,Z 686.308,A -85,B 0,C 180,E1 -22687.43,E2 -22687.43} C_VEL
LIN {X 0,Y 181.273,Z 686.488,A -85,B 0,C 180,E1 -22695.747,E2 -22695.747} C_VEL
LIN {X 0,Y 181.075,Z 687.274,A -85,B 0,C 180,E1 -22698.969,E2 -22698.969} C_VEL
LIN {X 0,Y 181.535,Z 689.47,A -85,B 0,C 180,E1 -22702.777,E2 -22702.777} C_VEL
LIN {X 0,Y 183.342,Z 694.019,A -85,B 0,C 180,E1 -22707.697,E2 -22707.697} C_VEL
LIN {X 0,Y 186.88,Z 699.73,A -85,B 0,C 180,E1 -22712.805,E2 -22712.805} C_VEL
LIN {X 0,Y 189.357,Z 705.654,A -85,B 0,C 180,E1 -22715.91,E2 -22715.91} C_VEL
LIN {X 0,Y 191.076,Z 708.418,A -85,B 0,C 180,E1 -22717.531,E2 -22717.531} C_VEL
LIN {X 0,Y 192.954,Z 713.518,A -85,B 0,C 180,E1 -22719.6,E2 -22719.6} C_VEL
LIN {X 0,Y 194.186,Z 715.801,A -85,B 0,C 180,E1 -22720.652,E2 -22720.652} C_VEL
LIN {X 0,Y 196.016,Z 720.795,A -85,B 0,C 180,E1 -22722.472,E2 -22722.472} C_VEL
LIN {X 0,Y 198.042,Z 726.757,A -85,B 0,C 180,E1 -22724.499,E2 -22724.499} C_VEL
LIN {X 0,Y 198.633,Z 734.625,A -85,B 0,C 180,E1 -22726.344,E2 -22726.344} C_VEL
LIN {X 0,Y 198.415,Z 746.783,A -85,B 0,C 180,E1 -22729.104,E2 -22729.104} C_VEL
LIN {X 0,Y 197.346,Z 757.349,A -85,B 0,C 180,E1 -22731.581,E2 -22731.581} C_VEL
LIN {X 0,Y 195.427,Z 767.776,A -85,B 0,C 180,E1 -22734.239,E2 -22734.239} C_VEL
LIN {X 0,Y 192.936,Z 777.115,A -85,B 0,C 180,E1 -22736.911,E2 -22736.911} C_VEL
LIN {X 0,Y 189.627,Z 786.339,A -85,B 0,C 180,E1 -22739.976,E2 -22739.976} C_VEL
LIN {X 0,Y 187.455,Z 792.897,A -85,B 0,C 180,E1 -22742.507,E2 -22742.507} C_VEL
LIN {X 0,Y 185.444,Z 802.638,A -85,B 0,C 180,E1 -22744.462,E2 -22744.462} C_VEL
LIN {X 0,Y 183.85,Z 809.864,A -85,B 0,C 180,E1 -22746.215,E2 -22746.215} C_VEL
LIN {X 0,Y 182.222,Z 814.221,A -85,B 0,C 180,E1 -22747.355,E2 -22747.355} C_VEL
LIN {X 0,Y 177.875,Z 820.78,A -85,B 0,C 180,E1 -22749.274,E2 -22749.274} C_VEL
LIN {X 0,Y 173.539,Z 826.74,A -85,B 0,C 180,E1 -22751.454,E2 -22751.454} C_VEL
LIN {X 0,Y 171.971,Z 830.166,A -85,B 0,C 180,E1 -22752.974,E2 -22752.974} C_VEL
LIN {X 0,Y 170.386,Z 837.516,A -85,B 0,C 180,E1 -22756.886,E2 -22756.886} C_VEL
LIN {X 0,Y 169.577,Z 842.706,A -85,B 0,C 180,E1 -22760.456,E2 -22760.456} C_VEL
LIN {X 0,Y 169.155,Z 846.678,A -85,B 0,C 180,E1 -22764.037,E2 -22764.037} C_VEL
LIN {X 0,Y 169.068,Z 849.561,A -85,B 0,C 180,E1 -22767.616,E2 -22767.616} C_VEL
LIN {X 0,Y 169.205,Z 850.904,A -85,B 0,C 180,E1 -22769.999,E2 -22769.999} C_VEL
LIN {X 0,Y 169.003,Z 852.336,A -85,B 0,C 180,E1 -22774.769,E2 -22774.769} C_VEL
LIN {X 0,Y 169.163,Z 852.478,A -85,B 0,C 180,E1 -22777.158,E2 -22777.158} C_VEL
LIN {X 0,Y 170.176,Z 851.542,A -85,B 0,C 180,E1 -22781.915,E2 -22781.915} C_VEL
LIN {X 0,Y 172.147,Z 849.11,A -85,B 0,C 180,E1 -22786.604,E2 -22786.604} C_VEL
LIN {X 0,Y 174.545,Z 846.221,A -85,B 0,C 180,E1 -22790.013,E2 -22790.013} C_VEL
LIN {X 0,Y 177.613,Z 842.367,A -85,B 0,C 180,E1 -22793.308,E2 -22793.308} C_VEL
LIN {X 0,Y 181.791,Z 836.23,A -85,B 0,C 180,E1 -22797.229,E2 -22797.229} C_VEL
LIN {X 0,Y 186.599,Z 829.111,A -85,B 0,C 180,E1 -22800.56,E2 -22800.56} C_VEL
LIN {X 0,Y 191.459,Z 821.21,A -85,B 0,C 180,E1 -22803.407,E2 -22803.407} C_VEL
LIN {X 0,Y 196.943,Z 811.397,A -85,B 0,C 180,E1 -22806.071,E2 -22806.071} C_VEL
LIN {X 0,Y 201.585,Z 800.603,A -85,B 0,C 180,E1 -22808.548,E2 -22808.548} C_VEL
LIN {X 0,Y 205.187,Z 789.981,A -85,B 0,C 180,E1 -22810.599,E2 -22810.599} C_VEL
LIN {X 0,Y 207.006,Z 780.666,A -85,B 0,C 180,E1 -22812.434,E2 -22812.434} C_VEL
LIN {X 0,Y 207.945,Z 770.166,A -85,B 0,C 180,E1 -22814.557,E2 -22814.557} C_VEL
LIN {X 0,Y 207.859,Z 760.639,A -85,B 0,C 180,E1 -22816.618,E2 -22816.618} C_VEL
LIN {X 0,Y 207.223,Z 753.16,A -85,B 0,C 180,E1 -22818.381,E2 -22818.381} C_VEL
LIN {X 0,Y 204.868,Z 747.275,A -85,B 0,C 180,E1 -22820.962,E2 -22820.962} C_VEL
LIN {X 0,Y 202.683,Z 742.021,A -85,B 0,C 180,E1 -22823.744,E2 -22823.744} C_VEL
LIN {X 0,Y 200.374,Z 739.201,A -85,B 0,C 180,E1 -22826.874,E2 -22826.874} C_VEL
LIN {X 0,Y 198.439,Z 737.314,A -85,B 0,C 180,E1 -22830.738,E2 -22830.738} C_VEL
LIN {X 0,Y 197.524,Z 736.86,A -85,B 0,C 180,E1 -22834.724,E2 -22834.724} C_VEL
LIN {X 0,Y 197.747,Z 738.442,A -85,B 0,C 180,E1 -22839.393,E2 -22839.393} C_VEL
LIN {X 0,Y 199.588,Z 741.814,A -85,B 0,C 180,E1 -22844.163,E2 -22844.163} C_VEL
LIN {X 0,Y 202.349,Z 747.545,A -85,B 0,C 180,E1 -22848.575,E2 -22848.575} C_VEL
LIN {X 0,Y 204.034,Z 751.891,A -85,B 0,C 180,E1 -22850.936,E2 -22850.936} C_VEL
LIN {X 0,Y 205.201,Z 755.439,A -85,B 0,C 180,E1 -22852.513,E2 -22852.513} C_VEL
LIN {X 0,Y 205.797,Z 760.625,A -85,B 0,C 180,E1 -22854.119,E2 -22854.119} C_VEL
LIN {X 0,Y 206.118,Z 771.465,A -85,B 0,C 180,E1 -22857.068,E2 -22857.068} C_VEL
LIN {X 0,Y 205.621,Z 780.743,A -85,B 0,C 180,E1 -22859.51,E2 -22859.51} C_VEL
LIN {X 0,Y 204.18,Z 790.258,A -85,B 0,C 180,E1 -22861.972,E2 -22861.972} C_VEL
LIN {X 0,Y 203.13,Z 794.717,A -85,B 0,C 180,E1 -22863.148,E2 -22863.148} C_VEL
LIN {X 0,Y 197.735,Z 805.846,A -85,B 0,C 180,E1 -22865.638,E2 -22865.638} C_VEL
LIN {X 0,Y 192.3,Z 815.352,A -85,B 0,C 180,E1 -22868.406,E2 -22868.406} C_VEL
LIN {X 0,Y 187.516,Z 822.866,A -85,B 0,C 180,E1 -22871.282,E2 -22871.282} C_VEL
LIN {X 0,Y 183.32,Z 828.793,A -85,B 0,C 180,E1 -22874.199,E2 -22874.199} C_VEL
LIN {X 0,Y 179.934,Z 833.27,A -85,B 0,C 180,E1 -22877.034,E2 -22877.034} C_VEL
LIN {X 0,Y 176.033,Z 837.997,A -85,B 0,C 180,E1 -22881.058,E2 -22881.058} C_VEL
LIN {X 0,Y 173.89,Z 840.284,A -85,B 0,C 180,E1 -22883.838,E2 -22883.838} C_VEL
LIN {X 0,Y 172.182,Z 841.976,A -85,B 0,C 180,E1 -22886.679,E2 -22886.679} C_VEL
LIN {X 0,Y 170.579,Z 843.213,A -85,B 0,C 180,E1 -22890.096,E2 -22890.096} C_VEL
LIN {X 0,Y 169.319,Z 843.609,A -85,B 0,C 180,E1 -22893.889,E2 -22893.889} C_VEL
LIN {X 0,Y 168.484,Z 842.644,A -85,B 0,C 180,E1 -22898.733,E2 -22898.733} C_VEL
LIN {X 0,Y 168.453,Z 840.246,A -85,B 0,C 180,E1 -22903.363,E2 -22903.363} C_VEL
LIN {X 0,Y 168.792,Z 837.482,A -85,B 0,C 180,E1 -22906.726,E2 -22906.726} C_VEL
LIN {X 0,Y 169.72,Z 832.814,A -85,B 0,C 180,E1 -22910.862,E2 -22910.862} C_VEL
LIN {X 0,Y 171.206,Z 826.152,A -85,B 0,C 180,E1 -22915.184,E2 -22915.184} C_VEL
LIN {X 0,Y 172.863,Z 819.291,A -85,B 0,C 180,E1 -22918.625,E2 -22918.625} C_VEL
LIN {X 0,Y 175.043,Z 810.624,A -85,B 0,C 180,E1 -22922.043,E2 -22922.043} C_VEL
LIN {X 0,Y 177.564,Z 800.591,A -85,B 0,C 180,E1 -22925.174,E2 -22925.174} C_VEL
LIN {X 0,Y 180.199,Z 789.447,A -85,B 0,C 180,E1 -22927.88,E2 -22927.88} C_VEL
LIN {X 0,Y 182.58,Z 778.221,A -85,B 0,C 180,E1 -22930.026,E2 -22930.026} C_VEL
LIN {X 0,Y 182.032,Z 766.929,A -85,B 0,C 180,E1 -22932.01,E2 -22932.01} C_VEL
LIN {X 0,Y 180.767,Z 753.777,A -85,B 0,C 180,E1 -22933.919,E2 -22933.919} C_VEL
LIN {X 0,Y 178.981,Z 740.438,A -85,B 0,C 180,E1 -22935.432,E2 -22935.432} C_VEL
LIN {X 0,Y 177.581,Z 732.565,A -85,B 0,C 180,E1 -22936.192,E2 -22936.192} C_VEL
LIN {X 0,Y 179.333,Z 723.146,A -85,B 0,C 180,E1 -22940.982,E2 -22940.982} C_VEL
LIN {X 0,Y 180.082,Z 718.737,A -85,B 0,C 180,E1 -22943.278,E2 -22943.278} C_VEL
LIN {X 0,Y 179.538,Z 712.868,A -85,B 0,C 180,E1 -22946.635,E2 -22946.635} C_VEL
LIN {X 0,Y 178.574,Z 705.285,A -85,B 0,C 180,E1 -22951.129,E2 -22951.129} C_VEL
LIN {X 0,Y 177.847,Z 701.654,A -85,B 0,C 180,E1 -22953.399,E2 -22953.399} C_VEL
LIN {X 0,Y 176.811,Z 697.764,A -85,B 0,C 180,E1 -22955.989,E2 -22955.989} C_VEL
LIN {X 0,Y 179.987,Z 701.495,A -85,B 0,C 180,E1 -22957.222,E2 -22957.222} C_VEL
LIN {X 0,Y 182.915,Z 712.001,A -85,B 0,C 180,E1 -22959.958,E2 -22959.958} C_VEL
LIN {X 0,Y 183.978,Z 716.698,A -85,B 0,C 180,E1 -22961.291,E2 -22961.291} C_VEL
LIN {X 0,Y 181.765,Z 726.757,A -85,B 0,C 180,E1 -22963.873,E2 -22963.873} C_VEL
LIN {X 0,Y 179.174,Z 736.762,A -85,B 0,C 180,E1 -22967.11,E2 -22967.11} C_VEL
LIN {X 0,Y 177.055,Z 744.727,A -85,B 0,C 180,E1 -22970.354,E2 -22970.354} C_VEL
LIN {X 0,Y 175.346,Z 751.157,A -85,B 0,C 180,E1 -22973.63,E2 -22973.63} C_VEL
LIN {X 0,Y 173.935,Z 756.776,A -85,B 0,C 180,E1 -22977.261,E2 -22977.261} C_VEL
LIN {X 0,Y 172.831,Z 761.578,A -85,B 0,C 180,E1 -22981.357,E2 -22981.357} C_VEL
LIN {X 0,Y 172.336,Z 764.928,A -85,B 0,C 180,E1 -22985.352,E2 -22985.352} C_VEL
LIN {X 0,Y 172.469,Z 767.044,A -85,B 0,C 180,E1 -22989.264,E2 -22989.264} C_VEL
LIN {X 0,Y 173.383,Z 768.091,A -85,B 0,C 180,E1 -22993.559,E2 -22993.559} C_VEL
LIN {X 0,Y 174.564,Z 767.998,A -85,B 0,C 180,E1 -22996.81,E2 -22996.81} C_VEL
LIN {X 0,Y 176.345,Z 766.988,A -85,B 0,C 180,E1 -23000.383,E2 -23000.383} C_VEL
LIN {X 0,Y 178.58,Z 765.058,A -85,B 0,C 180,E1 -23003.82,E2 -23003.82} C_VEL
LIN {X 0,Y 182.104,Z 761.143,A -85,B 0,C 180,E1 -23008.11,E2 -23008.11} C_VEL
LIN {X 0,Y 184.949,Z 757.5,A -85,B 0,C 180,E1 -23010.927,E2 -23010.927} C_VEL
LIN {X 0,Y 189.055,Z 751.554,A -85,B 0,C 180,E1 -23014.354,E2 -23014.354} C_VEL
LIN {X 0,Y 192.731,Z 745.52,A -85,B 0,C 180,E1 -23017.038,E2 -23017.038} C_VEL
LIN {X 0,Y 196.78,Z 738.085,A -85,B 0,C 180,E1 -23019.657,E2 -23019.657} C_VEL
LIN {X 0,Y 197.469,Z 736.356,A -85,B 0,C 180,E1 -23020.262,E2 -23020.262} C_VEL
LIN {X 0,Y 197.312,Z 730.652,A -85,B 0,C 180,E1 -23022.911,E2 -23022.911} C_VEL
LIN {X 0,Y 196.157,Z 722.959,A -85,B 0,C 180,E1 -23026.533,E2 -23026.533} C_VEL
LIN {X 0,Y 194.525,Z 716.726,A -85,B 0,C 180,E1 -23029.593,E2 -23029.593} C_VEL
LIN {X 0,Y 192.586,Z 710.976,A -85,B 0,C 180,E1 -23032.662,E2 -23032.662} C_VEL
LIN {X 0,Y 190.246,Z 705.57,A -85,B 0,C 180,E1 -23035.895,E2 -23035.895} C_VEL
LIN {X 0,Y 187.341,Z 699.799,A -85,B 0,C 180,E1 -23040,E2 -23040} C_VEL
LIN {X 0,Y 186.023,Z 696.955,A -85,B 0,C 180,E1 -23042.165,E2 -23042.165} C_VEL
LIN {X 0,Y 183.091,Z 694.084,A -85,B 0,C 180,E1 -23046.613,E2 -23046.613} C_VEL
LIN {X 0,Y 181.909,Z 693.125,A -85,B 0,C 180,E1 -23048.89,E2 -23048.89} C_VEL
LIN {X 0,Y 179.643,Z 693.436,A -85,B 0,C 180,E1 -23055.894,E2 -23055.894} C_VEL
LIN {X 0,Y 179.584,Z 694.522,A -85,B 0,C 180,E1 -23059.701,E2 -23059.701} C_VEL
LIN {X 0,Y 180.136,Z 697.173,A -85,B 0,C 180,E1 -23063.573,E2 -23063.573} C_VEL
LIN {X 0,Y 183.308,Z 704.314,A -85,B 0,C 180,E1 -23070.691,E2 -23070.691} C_VEL
LIN {X 0,Y 184.319,Z 706.054,A -85,B 0,C 180,E1 -23072.103,E2 -23072.103} C_VEL
LIN {X 0,Y 186.437,Z 711.76,A -85,B 0,C 180,E1 -23075.258,E2 -23075.258} C_VEL
LIN {X 0,Y 187.809,Z 714.399,A -85,B 0,C 180,E1 -23076.78,E2 -23076.78} C_VEL
LIN {X 0,Y 189.62,Z 719.506,A -85,B 0,C 180,E1 -23079.057,E2 -23079.057} C_VEL
LIN {X 0,Y 190.279,Z 720.787,A -85,B 0,C 180,E1 -23079.709,E2 -23079.709} C_VEL
LIN {X 0,Y 191.547,Z 725.114,A -85,B 0,C 180,E1 -23081.333,E2 -23081.333} C_VEL
LIN {X 0,Y 192.536,Z 728.168,A -85,B 0,C 180,E1 -23082.479,E2 -23082.479} C_VEL
LIN {X 0,Y 193.454,Z 731.416,A -85,B 0,C 180,E1 -23083.651,E2 -23083.651} C_VEL
LIN {X 0,Y 193.422,Z 742.37,A -85,B 0,C 180,E1 -23086.34,E2 -23086.34} C_VEL
LIN {X 0,Y 192.352,Z 754.001,A -85,B 0,C 180,E1 -23089.218,E2 -23089.218} C_VEL
LIN {X 0,Y 190.282,Z 765.125,A -85,B 0,C 180,E1 -23092.117,E2 -23092.117} C_VEL
LIN {X 0,Y 187.505,Z 775.429,A -85,B 0,C 180,E1 -23095.137,E2 -23095.137} C_VEL
LIN {X 0,Y 183.985,Z 784.741,A -85,B 0,C 180,E1 -23098.315,E2 -23098.315} C_VEL
LIN {X 0,Y 180.576,Z 793.511,A -85,B 0,C 180,E1 -23101.999,E2 -23101.999} C_VEL
LIN {X 0,Y 178.187,Z 804.223,A -85,B 0,C 180,E1 -23104.286,E2 -23104.286} C_VEL
LIN {X 0,Y 175.895,Z 814.09,A -85,B 0,C 180,E1 -23106.942,E2 -23106.942} C_VEL
LIN {X 0,Y 173.736,Z 822.825,A -85,B 0,C 180,E1 -23109.888,E2 -23109.888} C_VEL
LIN {X 0,Y 171.971,Z 830.166,A -85,B 0,C 180,E1 -23112.974,E2 -23112.974} C_VEL
LIN {X 0,Y 170.51,Z 833.419,A -85,B 0,C 180,E1 -23114.564,E2 -23114.564} C_VEL
LIN {X 0,Y 166.701,Z 838.09,A -85,B 0,C 180,E1 -23117.246,E2 -23117.246} C_VEL
LIN {X 0,Y 163.198,Z 842.081,A -85,B 0,C 180,E1 -23120.161,E2 -23120.161} C_VEL
LIN {X 0,Y 162.245,Z 844.263,A -85,B 0,C 180,E1 -23122.065,E2 -23122.065} C_VEL
LIN {X 0,Y 161.989,Z 848.141,A -85,B 0,C 180,E1 -23126.269,E2 -23126.269} C_VEL
LIN {X 0,Y 162.125,Z 850.473,A -85,B 0,C 180,E1 -23129.999,E2 -23129.999} C_VEL
LIN {X 0,Y 161.89,Z 851.639,A -85,B 0,C 180,E1 -23133.15,E2 -23133.15} C_VEL
LIN {X 0,Y 162.121,Z 852.245,A -85,B 0,C 180,E1 -23137.471,E2 -23137.471} C_VEL
LIN {X 0,Y 162.531,Z 852.077,A -85,B 0,C 180,E1 -23139.959,E2 -23139.959} C_VEL
LIN {X 0,Y 164.158,Z 850.545,A -85,B 0,C 180,E1 -23144.883,E2 -23144.883} C_VEL
LIN {X 0,Y 165.331,Z 849.218,A -85,B 0,C 180,E1 -23147.31,E2 -23147.31} C_VEL
LIN {X 0,Y 167.875,Z 846.471,A -85,B 0,C 180,E1 -23150.844,E2 -23150.844} C_VEL
LIN {X 0,Y 171.128,Z 842.778,A -85,B 0,C 180,E1 -23154.246,E2 -23154.246} C_VEL
LIN {X 0,Y 175.353,Z 837.155,A -85,B 0,C 180,E1 -23158.146,E2 -23158.146} C_VEL
LIN {X 0,Y 180.581,Z 830.036,A -85,B 0,C 180,E1 -23161.694,E2 -23161.694} C_VEL
LIN {X 0,Y 184.715,Z 823.776,A -85,B 0,C 180,E1 -23164.137,E2 -23164.137} C_VEL
LIN {X 0,Y 190.44,Z 814.665,A -85,B 0,C 180,E1 -23166.846,E2 -23166.846} C_VEL
LIN {X 0,Y 194.893,Z 805.678,A -85,B 0,C 180,E1 -23169.127,E2 -23169.127} C_VEL
LIN {X 0,Y 199.146,Z 795.51,A -85,B 0,C 180,E1 -23171.254,E2 -23171.254} C_VEL
LIN {X 0,Y 201.231,Z 788.572,A -85,B 0,C 180,E1 -23172.641,E2 -23172.641} C_VEL
LIN {X 0,Y 202.951,Z 780.203,A -85,B 0,C 180,E1 -23174.394,E2 -23174.394} C_VEL
LIN {X 0,Y 203.916,Z 770.858,A -85,B 0,C 180,E1 -23176.425,E2 -23176.425} C_VEL
LIN {X 0,Y 204.058,Z 760.765,A -85,B 0,C 180,E1 -23178.802,E2 -23178.802} C_VEL
LIN {X 0,Y 203.825,Z 758.099,A -85,B 0,C 180,E1 -23179.547,E2 -23179.547} C_VEL
LIN {X 0,Y 202.189,Z 753.036,A -85,B 0,C 180,E1 -23181.88,E2 -23181.88} C_VEL
LIN {X 0,Y 200.53,Z 748.387,A -85,B 0,C 180,E1 -23184.443,E2 -23184.443} C_VEL
LIN {X 0,Y 198.668,Z 745.964,A -85,B 0,C 180,E1 -23187.274,E2 -23187.274} C_VEL
LIN {X 0,Y 196.888,Z 744.179,A -85,B 0,C 180,E1 -23191.191,E2 -23191.191} C_VEL
LIN {X 0,Y 196.097,Z 743.897,A -85,B 0,C 180,E1 -23195.107,E2 -23195.107} C_VEL
LIN {X 0,Y 196.323,Z 745.632,A -85,B 0,C 180,E1 -23199.661,E2 -23199.661} C_VEL
LIN {X 0,Y 197.664,Z 748.488,A -85,B 0,C 180,E1 -23203.733,E2 -23203.733} C_VEL
LIN {X 0,Y 199.759,Z 753.794,A -85,B 0,C 180,E1 -23207.925,E2 -23207.925} C_VEL
LIN {X 0,Y 201.189,Z 758.237,A -85,B 0,C 180,E1 -23210.447,E2 -23210.447} C_VEL
LIN {X 0,Y 201.912,Z 761.914,A -85,B 0,C 180,E1 -23211.996,E2 -23211.996} C_VEL
LIN {X 0,Y 201.936,Z 771.266,A -85,B 0,C 180,E1 -23214.789,E2 -23214.789} C_VEL
LIN {X 0,Y 201.284,Z 780.866,A -85,B 0,C 180,E1 -23217.498,E2 -23217.498} C_VEL
LIN {X 0,Y 199.75,Z 789.951,A -85,B 0,C 180,E1 -23220,E2 -23220} C_VEL
LIN {X 0,Y 198.136,Z 796.214,A -85,B 0,C 180,E1 -23221.723,E2 -23221.723} C_VEL
LIN {X 0,Y 194.539,Z 803.505,A -85,B 0,C 180,E1 -23223.364,E2 -23223.364} C_VEL
LIN {X 0,Y 188.777,Z 813.344,A -85,B 0,C 180,E1 -23226.067,E2 -23226.067} C_VEL
LIN {X 0,Y 183.761,Z 820.966,A -85,B 0,C 180,E1 -23228.799,E2 -23228.799} C_VEL
LIN {X 0,Y 179.356,Z 827.047,A -85,B 0,C 180,E1 -23231.597,E2 -23231.597} C_VEL
LIN {X 0,Y 174.696,Z 832.828,A -85,B 0,C 180,E1 -23235.096,E2 -23235.096} C_VEL
LIN {X 0,Y 170.264,Z 837.778,A -85,B 0,C 180,E1 -23239.282,E2 -23239.282} C_VEL
LIN {X 0,Y 167.507,Z 840.525,A -85,B 0,C 180,E1 -23242.63,E2 -23242.63} C_VEL
LIN {X 0,Y 165.044,Z 842.645,A -85,B 0,C 180,E1 -23246.594,E2 -23246.594} C_VEL
LIN {X 0,Y 163.015,Z 843.764,A -85,B 0,C 180,E1 -23251.154,E2 -23251.154} C_VEL
LIN {X 0,Y 162.055,Z 843.703,A -85,B 0,C 180,E1 -23254.516,E2 -23254.516} C_VEL
LIN {X 0,Y 161.41,Z 842.769,A -85,B 0,C 180,E1 -23258.398,E2 -23258.398} C_VEL
LIN {X 0,Y 161.304,Z 840.916,A -85,B 0,C 180,E1 -23262.212,E2 -23262.212} C_VEL
LIN {X 0,Y 161.578,Z 838.195,A -85,B 0,C 180,E1 -23265.901,E2 -23265.901} C_VEL
LIN {X 0,Y 162.253,Z 834.596,A -85,B 0,C 180,E1 -23269.481,E2 -23269.481} C_VEL
LIN {X 0,Y 163.495,Z 828.755,A -85,B 0,C 180,E1 -23273.854,E2 -23273.854} C_VEL
LIN {X 0,Y 164.987,Z 822.779,A -85,B 0,C 180,E1 -23277.306,E2 -23277.306} C_VEL
LIN {X 0,Y 166.836,Z 815.419,A -85,B 0,C 180,E1 -23280.703,E2 -23280.703} C_VEL
LIN {X 0,Y 169.192,Z 806.372,A -85,B 0,C 180,E1 -23284.031,E2 -23284.031} C_VEL
LIN {X 0,Y 171.672,Z 796.947,A -85,B 0,C 180,E1 -23286.796,E2 -23286.796} C_VEL
LIN {X 0,Y 174.282,Z 785.937,A -85,B 0,C 180,E1 -23289.34,E2 -23289.34} C_VEL
LIN {X 0,Y 175.819,Z 778.572,A -85,B 0,C 180,E1 -23290.746,E2 -23290.746} C_VEL
LIN {X 0,Y 175.305,Z 767.399,A -85,B 0,C 180,E1 -23292.804,E2 -23292.804} C_VEL
LIN {X 0,Y 174.13,Z 754.172,A -85,B 0,C 180,E1 -23294.792,E2 -23294.792} C_VEL
LIN {X 0,Y 172.348,Z 740.914,A -85,B 0,C 180,E1 -23296.366,E2 -23296.366} C_VEL
LIN {X 0,Y 170.933,Z 732.63,A -85,B 0,C 180,E1 -23297.234,E2 -23297.234} C_VEL
LIN {X 0,Y 172.933,Z 722.729,A -85,B 0,C 180,E1 -23302.411,E2 -23302.411} C_VEL
LIN {X 0,Y 173.27,Z 719.501,A -85,B 0,C 180,E1 -23304.181,E2 -23304.181} C_VEL
LIN {X 0,Y 172.611,Z 713.629,A -85,B 0,C 180,E1 -23307.668,E2 -23307.668} C_VEL
LIN {X 0,Y 171.684,Z 706.055,A -85,B 0,C 180,E1 -23312.347,E2 -23312.347} C_VEL
LIN {X 0,Y 170.499,Z 701.373,A -85,B 0,C 180,E1 -23315.574,E2 -23315.574} C_VEL
LIN {X 0,Y 173.767,Z 705.272,A -85,B 0,C 180,E1 -23316.97,E2 -23316.97} C_VEL
LIN {X 0,Y 175.506,Z 711.004,A -85,B 0,C 180,E1 -23318.566,E2 -23318.566} C_VEL
LIN {X 0,Y 177.225,Z 718.841,A -85,B 0,C 180,E1 -23320.859,E2 -23320.859} C_VEL
LIN {X 0,Y 174.65,Z 729.165,A -85,B 0,C 180,E1 -23323.676,E2 -23323.676} C_VEL
LIN {X 0,Y 172.299,Z 737.752,A -85,B 0,C 180,E1 -23326.591,E2 -23326.591} C_VEL
LIN {X 0,Y 170.113,Z 745.655,A -85,B 0,C 180,E1 -23329.929,E2 -23329.929} C_VEL
LIN {X 0,Y 168.35,Z 752.057,A -85,B 0,C 180,E1 -23333.305,E2 -23333.305} C_VEL
LIN {X 0,Y 166.724,Z 758.396,A -85,B 0,C 180,E1 -23337.627,E2 -23337.627} C_VEL
LIN {X 0,Y 165.653,Z 763.125,A -85,B 0,C 180,E1 -23341.949,E2 -23341.949} C_VEL
LIN {X 0,Y 165.275,Z 766.575,A -85,B 0,C 180,E1 -23346.537,E2 -23346.537} C_VEL
LIN {X 0,Y 165.558,Z 768.297,A -85,B 0,C 180,E1 -23350.173,E2 -23350.173} C_VEL
LIN {X 0,Y 166.499,Z 769.163,A -85,B 0,C 180,E1 -23354.145,E2 -23354.145} C_VEL
LIN {X 0,Y 168.358,Z 768.85,A -85,B 0,C 180,E1 -23358.713,E2 -23358.713} C_VEL
LIN {X 0,Y 170.06,Z 767.88,A -85,B 0,C 180,E1 -23361.741,E2 -23361.741} C_VEL
LIN {X 0,Y 173.377,Z 764.996,A -85,B 0,C 180,E1 -23366.351,E2 -23366.351} C_VEL
LIN {X 0,Y 176.192,Z 761.947,A -85,B 0,C 180,E1 -23369.507,E2 -23369.507} C_VEL
LIN {X 0,Y 179.482,Z 757.985,A -85,B 0,C 180,E1 -23372.529,E2 -23372.529} C_VEL
LIN {X 0,Y 183.128,Z 753.024,A -85,B 0,C 180,E1 -23375.467,E2 -23375.467} C_VEL
LIN {X 0,Y 188.221,Z 745.161,A -85,B 0,C 180,E1 -23378.986,E2 -23378.986} C_VEL
LIN {X 0,Y 190.899,Z 740.464,A -85,B 0,C 180,E1 -23380.65,E2 -23380.65} C_VEL
LIN {X 0,Y 191.612,Z 738.772,A -85,B 0,C 180,E1 -23381.281,E2 -23381.281} C_VEL
LIN {X 0,Y 191.558,Z 733.137,A -85,B 0,C 180,E1 -23384.115,E2 -23384.115} C_VEL
LIN {X 0,Y 190.861,Z 727.079,A -85,B 0,C 180,E1 -23387.236,E2 -23387.236} C_VEL
LIN {X 0,Y 189.612,Z 721.175,A -85,B 0,C 180,E1 -23390.399,E2 -23390.399} C_VEL
LIN {X 0,Y 188.009,Z 715.684,A -85,B 0,C 180,E1 -23393.561,E2 -23393.561} C_VEL
LIN {X 0,Y 186.189,Z 710.814,A -85,B 0,C 180,E1 -23396.755,E2 -23396.755} C_VEL
LIN {X 0,Y 183.201,Z 703.835,A -85,B 0,C 180,E1 -23402.199,E2 -23402.199} C_VEL
LIN {X 0,Y 182.941,Z 703.185,A -85,B 0,C 180,E1 -23402.752,E2 -23402.752} C_VEL
LIN {X 0,Y 180.703,Z 700.815,A -85,B 0,C 180,E1 -23406.701,E2 -23406.701} C_VEL
LIN {X 0,Y 179.704,Z 699.881,A -85,B 0,C 180,E1 -23409,E2 -23409} C_VEL
LIN {X 0,Y 177.647,Z 700.289,A -85,B 0,C 180,E1 -23416.078,E2 -23416.078} C_VEL
LIN {X 0,Y 177.563,Z 700.921,A -85,B 0,C 180,E1 -23418.46,E2 -23418.46} C_VEL
LIN {X 0,Y 177.697,Z 702.108,A -85,B 0,C 180,E1 -23420.852,E2 -23420.852} C_VEL
LIN {X 0,Y 178.628,Z 706.091,A -85,B 0,C 180,E1 -23425.645,E2 -23425.645} C_VEL
LIN {X 0,Y 180.828,Z 710.94,A -85,B 0,C 180,E1 -23430.349,E2 -23430.349} C_VEL
LIN {X 0,Y 181.733,Z 713.417,A -85,B 0,C 180,E1 -23432.059,E2 -23432.059} C_VEL
LIN {X 0,Y 184.392,Z 720.524,A -85,B 0,C 180,E1 -23436.214,E2 -23436.214} C_VEL
LIN {X 0,Y 186.169,Z 725.749,A -85,B 0,C 180,E1 -23438.724,E2 -23438.724} C_VEL
LIN {X 0,Y 188.056,Z 732.872,A -85,B 0,C 180,E1 -23441.63,E2 -23441.63} C_VEL
LIN {X 0,Y 188.696,Z 735.965,A -85,B 0,C 180,E1 -23442.774,E2 -23442.774} C_VEL
LIN {X 0,Y 188.031,Z 746.297,A -85,B 0,C 180,E1 -23445.481,E2 -23445.481} C_VEL
LIN {X 0,Y 186.487,Z 757.358,A -85,B 0,C 180,E1 -23448.429,E2 -23448.429} C_VEL
LIN {X 0,Y 184.342,Z 766.539,A -85,B 0,C 180,E1 -23451.018,E2 -23451.018} C_VEL
LIN {X 0,Y 181,Z 777.173,A -85,B 0,C 180,E1 -23454.377,E2 -23454.377} C_VEL
LIN {X 0,Y 177.911,Z 784.641,A -85,B 0,C 180,E1 -23457.1,E2 -23457.1} C_VEL
LIN {X 0,Y 174.541,Z 792.219,A -85,B 0,C 180,E1 -23460.444,E2 -23460.444} C_VEL
LIN {X 0,Y 173.644,Z 794.454,A -85,B 0,C 180,E1 -23461.52,E2 -23461.52} C_VEL
LIN {X 0,Y 170.97,Z 805.816,A -85,B 0,C 180,E1 -23464.102,E2 -23464.102} C_VEL
LIN {X 0,Y 168.864,Z 814.317,A -85,B 0,C 180,E1 -23466.537,E2 -23466.537} C_VEL
LIN {X 0,Y 166.639,Z 823.04,A -85,B 0,C 180,E1 -23469.637,E2 -23469.637} C_VEL
LIN {X 0,Y 164.65,Z 831.102,A -85,B 0,C 180,E1 -23473.253,E2 -23473.253} C_VEL
LIN {X 0,Y 163.425,Z 836.57,A -85,B 0,C 180,E1 -23476.317,E2 -23476.317} C_VEL
LIN {X 0,Y 162.552,Z 841.899,A -85,B 0,C 180,E1 -23480.04,E2 -23480.04} C_VEL
LIN {X 0,Y 162.245,Z 844.263,A -85,B 0,C 180,E1 -23482.065,E2 -23482.065} C_VEL
LIN {X 0,Y 161.385,Z 846.258,A -85,B 0,C 180,E1 -23484.013,E2 -23484.013} C_VEL
LIN {X 0,Y 159.718,Z 847.901,A -85,B 0,C 180,E1 -23485.966,E2 -23485.966} C_VEL
LIN {X 0,Y 155.981,Z 850.226,A -85,B 0,C 180,E1 -23490.029,E2 -23490.029} C_VEL
LIN {X 0,Y 154.813,Z 851.172,A -85,B 0,C 180,E1 -23492.926,E2 -23492.926} C_VEL
LIN {X 0,Y 155.057,Z 852.005,A -85,B 0,C 180,E1 -23497.814,E2 -23497.814} C_VEL
LIN {X 0,Y 156.273,Z 851.443,A -85,B 0,C 180,E1 -23502.993,E2 -23502.993} C_VEL
LIN {X 0,Y 158.544,Z 849.326,A -85,B 0,C 180,E1 -23508.076,E2 -23508.076} C_VEL
LIN {X 0,Y 162.336,Z 845.69,A -85,B 0,C 180,E1 -23512.93,E2 -23512.93} C_VEL
LIN {X 0,Y 165.924,Z 841.844,A -85,B 0,C 180,E1 -23516.405,E2 -23516.405} C_VEL
LIN {X 0,Y 168.977,Z 838.01,A -85,B 0,C 180,E1 -23519.14,E2 -23519.14} C_VEL
LIN {X 0,Y 174.639,Z 830.965,A -85,B 0,C 180,E1 -23522.905,E2 -23522.905} C_VEL
LIN {X 0,Y 179.924,Z 823.627,A -85,B 0,C 180,E1 -23525.866,E2 -23525.866} C_VEL
LIN {X 0,Y 185.918,Z 814.545,A -85,B 0,C 180,E1 -23528.587,E2 -23528.587} C_VEL
LIN {X 0,Y 191.545,Z 803.641,A -85,B 0,C 180,E1 -23531.331,E2 -23531.331} C_VEL
LIN {X 0,Y 195.608,Z 794.029,A -85,B 0,C 180,E1 -23533.351,E2 -23533.351} C_VEL
LIN {X 0,Y 197.984,Z 785.491,A -85,B 0,C 180,E1 -23535.229,E2 -23535.229} C_VEL
LIN {X 0,Y 199.576,Z 776.563,A -85,B 0,C 180,E1 -23537.238,E2 -23537.238} C_VEL
LIN {X 0,Y 200.411,Z 767.138,A -85,B 0,C 180,E1 -23539.523,E2 -23539.523} C_VEL
LIN {X 0,Y 200.497,Z 763.56,A -85,B 0,C 180,E1 -23540.456,E2 -23540.456} C_VEL
LIN {X 0,Y 199.246,Z 758.4,A -85,B 0,C 180,E1 -23542.948,E2 -23542.948} C_VEL
LIN {X 0,Y 198.249,Z 754.918,A -85,B 0,C 180,E1 -23544.948,E2 -23544.948} C_VEL
LIN {X 0,Y 196.722,Z 752.714,A -85,B 0,C 180,E1 -23547.596,E2 -23547.596} C_VEL
LIN {X 0,Y 195.305,Z 751.158,A -85,B 0,C 180,E1 -23550.935,E2 -23550.935} C_VEL
LIN {X 0,Y 194.501,Z 750.703,A -85,B 0,C 180,E1 -23554.597,E2 -23554.597} C_VEL
LIN {X 0,Y 194.43,Z 752.128,A -85,B 0,C 180,E1 -23558.809,E2 -23558.809} C_VEL
LIN {X 0,Y 195.412,Z 754.924,A -85,B 0,C 180,E1 -23563.157,E2 -23563.157} C_VEL
LIN {X 0,Y 196.677,Z 758.978,A -85,B 0,C 180,E1 -23566.608,E2 -23566.608} C_VEL
LIN {X 0,Y 197.992,Z 764.193,A -85,B 0,C 180,E1 -23569.777,E2 -23569.777} C_VEL
LIN {X 0,Y 198.295,Z 766.483,A -85,B 0,C 180,E1 -23570.819,E2 -23570.819} C_VEL
LIN {X 0,Y 197.865,Z 774.724,A -85,B 0,C 180,E1 -23573.434,E2 -23573.434} C_VEL
LIN {X 0,Y 196.583,Z 784.664,A -85,B 0,C 180,E1 -23576.413,E2 -23576.413} C_VEL
LIN {X 0,Y 194.614,Z 793.444,A -85,B 0,C 180,E1 -23578.965,E2 -23578.965} C_VEL
LIN {X 0,Y 193.046,Z 798.483,A -85,B 0,C 180,E1 -23580.439,E2 -23580.439} C_VEL
LIN {X 0,Y 187.172,Z 808.853,A -85,B 0,C 180,E1 -23582.959,E2 -23582.959} C_VEL
LIN {X 0,Y 181.608,Z 817.32,A -85,B 0,C 180,E1 -23585.611,E2 -23585.611} C_VEL
LIN {X 0,Y 176.462,Z 824.288,A -85,B 0,C 180,E1 -23588.453,E2 -23588.453} C_VEL
LIN {X 0,Y 171.251,Z 830.563,A -85,B 0,C 180,E1 -23591.841,E2 -23591.841} C_VEL
LIN {X 0,Y 166.067,Z 836.231,A -85,B 0,C 180,E1 -23596.057,E2 -23596.057} C_VEL
LIN {X 0,Y 162.021,Z 840.101,A -85,B 0,C 180,E1 -23600.305,E2 -23600.305} C_VEL
LIN {X 0,Y 159.757,Z 841.954,A -85,B 0,C 180,E1 -23603.323,E2 -23603.323} C_VEL
LIN {X 0,Y 157.661,Z 843.371,A -85,B 0,C 180,E1 -23606.938,E2 -23606.938} C_VEL
LIN {X 0,Y 155.89,Z 844.02,A -85,B 0,C 180,E1 -23611.069,E2 -23611.069} C_VEL
LIN {X 0,Y 154.604,Z 843.457,A -85,B 0,C 180,E1 -23616.224,E2 -23616.224} C_VEL
LIN {X 0,Y 154.219,Z 842.21,A -85,B 0,C 180,E1 -23619.643,E2 -23619.643} C_VEL
LIN {X 0,Y 154.352,Z 838.996,A -85,B 0,C 180,E1 -23624.888,E2 -23624.888} C_VEL
LIN {X 0,Y 154.961,Z 835.691,A -85,B 0,C 180,E1 -23628.544,E2 -23628.544} C_VEL
LIN {X 0,Y 155.915,Z 831.025,A -85,B 0,C 180,E1 -23632.462,E2 -23632.462} C_VEL
LIN {X 0,Y 157.629,Z 824.1,A -85,B 0,C 180,E1 -23636.899,E2 -23636.899} C_VEL
LIN {X 0,Y 159.295,Z 817.488,A -85,B 0,C 180,E1 -23640.243,E2 -23640.243} C_VEL
LIN {X 0,Y 161.494,Z 809.496,A -85,B 0,C 180,E1 -23643.51,E2 -23643.51} C_VEL
LIN {X 0,Y 164.101,Z 799.782,A -85,B 0,C 180,E1 -23646.664,E2 -23646.664} C_VEL
LIN {X 0,Y 166.97,Z 788.476,A -85,B 0,C 180,E1 -23649.552,E2 -23649.552} C_VEL
LIN {X 0,Y 169.018,Z 778.819,A -85,B 0,C 180,E1 -23651.516,E2 -23651.516} C_VEL
LIN {X 0,Y 168.49,Z 765.819,A -85,B 0,C 180,E1 -23653.958,E2 -23653.958} C_VEL
LIN {X 0,Y 167.339,Z 753.479,A -85,B 0,C 180,E1 -23655.872,E2 -23655.872} C_VEL
LIN {X 0,Y 165.503,Z 739.846,A -85,B 0,C 180,E1 -23657.533,E2 -23657.533} C_VEL
LIN {X 0,Y 164.312,Z 732.817,A -85,B 0,C 180,E1 -23658.276,E2 -23658.276} C_VEL
LIN {X 0,Y 166.315,Z 723.438,A -85,B 0,C 180,E1 -23663.328,E2 -23663.328} C_VEL
LIN {X 0,Y 166.411,Z 720.243,A -85,B 0,C 180,E1 -23665.156,E2 -23665.156} C_VEL
LIN {X 0,Y 165.51,Z 712.486,A -85,B 0,C 180,E1 -23670.001,E2 -23670.001} C_VEL
LIN {X 0,Y 165.083,Z 708.717,A -85,B 0,C 180,E1 -23672.441,E2 -23672.441} C_VEL
LIN {X 0,Y 164.149,Z 704.896,A -85,B 0,C 180,E1 -23675.168,E2 -23675.168} C_VEL
LIN {X 0,Y 167.659,Z 709.076,A -85,B 0,C 180,E1 -23676.771,E2 -23676.771} C_VEL
LIN {X 0,Y 169.227,Z 714.312,A -85,B 0,C 180,E1 -23678.359,E2 -23678.359} C_VEL
LIN {X 0,Y 170.444,Z 719.893,A -85,B 0,C 180,E1 -23680.094,E2 -23680.094} C_VEL
LIN {X 0,Y 167.912,Z 730.119,A -85,B 0,C 180,E1 -23683.002,E2 -23683.002} C_VEL
LIN {X 0,Y 165.455,Z 738.728,A -85,B 0,C 180,E1 -23686.029,E2 -23686.029} C_VEL
LIN {X 0,Y 163.205,Z 746.595,A -85,B 0,C 180,E1 -23689.478,E2 -23689.478} C_VEL
LIN {X 0,Y 161.08,Z 754.006,A -85,B 0,C 180,E1 -23693.618,E2 -23693.618} C_VEL
LIN {X 0,Y 159.448,Z 760.206,A -85,B 0,C 180,E1 -23698.172,E2 -23698.172} C_VEL
LIN {X 0,Y 158.494,Z 764.644,A -85,B 0,C 180,E1 -23702.595,E2 -23702.595} C_VEL
LIN {X 0,Y 158.23,Z 767.662,A -85,B 0,C 180,E1 -23706.919,E2 -23706.919} C_VEL
LIN {X 0,Y 158.764,Z 769.629,A -85,B 0,C 180,E1 -23711.607,E2 -23711.607} C_VEL
LIN {X 0,Y 159.827,Z 770.254,A -85,B 0,C 180,E1 -23715.287,E2 -23715.287} C_VEL
LIN {X 0,Y 161.524,Z 770.001,A -85,B 0,C 180,E1 -23719.258,E2 -23719.258} C_VEL
LIN {X 0,Y 164.564,Z 768.244,A -85,B 0,C 180,E1 -23724.237,E2 -23724.237} C_VEL
LIN {X 0,Y 168.222,Z 765.021,A -85,B 0,C 180,E1 -23728.773,E2 -23728.773} C_VEL
LIN {X 0,Y 171.349,Z 761.778,A -85,B 0,C 180,E1 -23731.867,E2 -23731.867} C_VEL
LIN {X 0,Y 175.711,Z 756.558,A -85,B 0,C 180,E1 -23735.498,E2 -23735.498} C_VEL
LIN {X 0,Y 180.685,Z 749.75,A -85,B 0,C 180,E1 -23738.991,E2 -23738.991} C_VEL
LIN {X 0,Y 185.062,Z 742.848,A -85,B 0,C 180,E1 -23741.7,E2 -23741.7} C_VEL
LIN {X 0,Y 185.767,Z 741.158,A -85,B 0,C 180,E1 -23742.383,E2 -23742.383} C_VEL
LIN {X 0,Y 185.836,Z 735.061,A -85,B 0,C 180,E1 -23745.77,E2 -23745.77} C_VEL
LIN {X 0,Y 185.314,Z 729.172,A -85,B 0,C 180,E1 -23749.069,E2 -23749.069} C_VEL
LIN {X 0,Y 184.25,Z 723.726,A -85,B 0,C 180,E1 -23752.328,E2 -23752.328} C_VEL
LIN {X 0,Y 182.968,Z 718.756,A -85,B 0,C 180,E1 -23755.594,E2 -23755.594} C_VEL
LIN {X 0,Y 180.57,Z 711.853,A -85,B 0,C 180,E1 -23761.017,E2 -23761.017} C_VEL
LIN {X 0,Y 180.075,Z 710.451,A -85,B 0,C 180,E1 -23762.237,E2 -23762.237} C_VEL
LIN {X 0,Y 179.039,Z 708.651,A -85,B 0,C 180,E1 -23764.503,E2 -23764.503} C_VEL
LIN {X 0,Y 177.463,Z 706.854,A -85,B 0,C 180,E1 -23768.077,E2 -23768.077} C_VEL
LIN {X 0,Y 177.111,Z 706.516,A -85,B 0,C 180,E1 -23769.133,E2 -23769.133} C_VEL
LIN {X 0,Y 175.306,Z 707.052,A -85,B 0,C 180,E1 -23776.298,E2 -23776.298} C_VEL
LIN {X 0,Y 175.243,Z 707.841,A -85,B 0,C 180,E1 -23778.714,E2 -23778.714} C_VEL
LIN {X 0,Y 175.58,Z 710.562,A -85,B 0,C 180,E1 -23782.98,E2 -23782.98} C_VEL
LIN {X 0,Y 177.724,Z 716.888,A -85,B 0,C 180,E1 -23789.542,E2 -23789.542} C_VEL
LIN {X 0,Y 178.485,Z 719.365,A -85,B 0,C 180,E1 -23791.36,E2 -23791.36} C_VEL
LIN {X 0,Y 180.481,Z 725.44,A -85,B 0,C 180,E1 -23795.139,E2 -23795.139} C_VEL
LIN {X 0,Y 182.1,Z 731.422,A -85,B 0,C 180,E1 -23798.135,E2 -23798.135} C_VEL
LIN {X 0,Y 183.583,Z 738.503,A -85,B 0,C 180,E1 -23801.2,E2 -23801.2} C_VEL
LIN {X 0,Y 183.768,Z 739.964,A -85,B 0,C 180,E1 -23801.751,E2 -23801.751} C_VEL
LIN {X 0,Y 182.749,Z 749.106,A -85,B 0,C 180,E1 -23804.305,E2 -23804.305} C_VEL
LIN {X 0,Y 180.624,Z 760.192,A -85,B 0,C 180,E1 -23807.501,E2 -23807.501} C_VEL
LIN {X 0,Y 177.577,Z 770.63,A -85,B 0,C 180,E1 -23810.71,E2 -23810.71} C_VEL
LIN {X 0,Y 173.871,Z 780.355,A -85,B 0,C 180,E1 -23814.145,E2 -23814.145} C_VEL
LIN {X 0,Y 169.952,Z 788.414,A -85,B 0,C 180,E1 -23817.479,E2 -23817.479} C_VEL
LIN {X 0,Y 166.714,Z 795.279,A -85,B 0,C 180,E1 -23821,E2 -23821} C_VEL
LIN {X 0,Y 164.031,Z 806.134,A -85,B 0,C 180,E1 -23823.606,E2 -23823.606} C_VEL
LIN {X 0,Y 161.685,Z 815.013,A -85,B 0,C 180,E1 -23826.305,E2 -23826.305} C_VEL
LIN {X 0,Y 159.551,Z 823.144,A -85,B 0,C 180,E1 -23829.365,E2 -23829.365} C_VEL
LIN {X 0,Y 157.523,Z 831.146,A -85,B 0,C 180,E1 -23833.141,E2 -23833.141} C_VEL
LIN {X 0,Y 156.134,Z 837.569,A -85,B 0,C 180,E1 -23836.992,E2 -23836.992} C_VEL
LIN {X 0,Y 155.342,Z 842.627,A -85,B 0,C 180,E1 -23840.888,E2 -23840.888} C_VEL
LIN {X 0,Y 154.99,Z 846.497,A -85,B 0,C 180,E1 -23844.795,E2 -23844.795} C_VEL
LIN {X 0,Y 154.906,Z 848.454,A -85,B 0,C 180,E1 -23847.398,E2 -23847.398} C_VEL
LIN {X 0,Y 155.045,Z 849.991,A -85,B 0,C 180,E1 -23849.999,E2 -23849.999} C_VEL
LIN {X 0,Y 154.813,Z 851.172,A -85,B 0,C 180,E1 -23852.926,E2 -23852.926} C_VEL
LIN {X 0,Y 154.148,Z 851.682,A -85,B 0,C 180,E1 -23855.097,E2 -23855.097} C_VEL
LIN {X 0,Y 151.64,Z 851.905,A -85,B 0,C 180,E1 -23858.692,E2 -23858.692} C_VEL
LIN {X 0,Y 149.855,Z 851.692,A -85,B 0,C 180,E1 -23861.646,E2 -23861.646} C_VEL
LIN {X 0,Y 149.525,Z 851.283,A -85,B 0,C 180,E1 -23863.909,E2 -23863.909} C_VEL
LIN {X 0,Y 149.722,Z 851.049,A -85,B 0,C 180,E1 -23864.66,E2 -23864.66} C_VEL
LIN {X 0,Y 151.794,Z 849.464,A -85,B 0,C 180,E1 -23868.909,E2 -23868.909} C_VEL
